REGION Network 64: **** 5.2 - Flow Equations **** Send Alarm If No Other Requests Is Active
   // Send Alarm If No Other Requests Is Active
   IF #SendAlarm[9] THEN
       #ReqSendToVDAlarm[9] := TRUE;   // SR flip-flop
   END_IF;
   IF #SendDoneVD THEN #ReqSendToVDAlarm[9] := FALSE; END_IF;
   IF #SendAlarm[9] THEN
       #_LDBCheckMZ8(I_DBNr := #C_AlarmDBMZ8, O_DBLength => #AlarmLength, O_DBNr => #AlarmPointer);   // "LDBCheck"
   END_IF;
   IF "TRUE" THEN
       #_LMDBToDBMZ8(I_CopyDB := #SendAlarm[9],   // "LMDBToDB"
                     I_SourceDB := #C_AlarmDBMZ8,
                     I_StartAddresSourceDB := 0,
                     I_DestDB := #C_AlarmCompareDBMZ8,
                     I_StartAddressDestDB := 0,
                     I_LenghtBytes := #AlarmLength);
   END_IF;
END_REGION

REGION Network 65: **** 5.2 - Flow Equations **** Filter
   // Filter
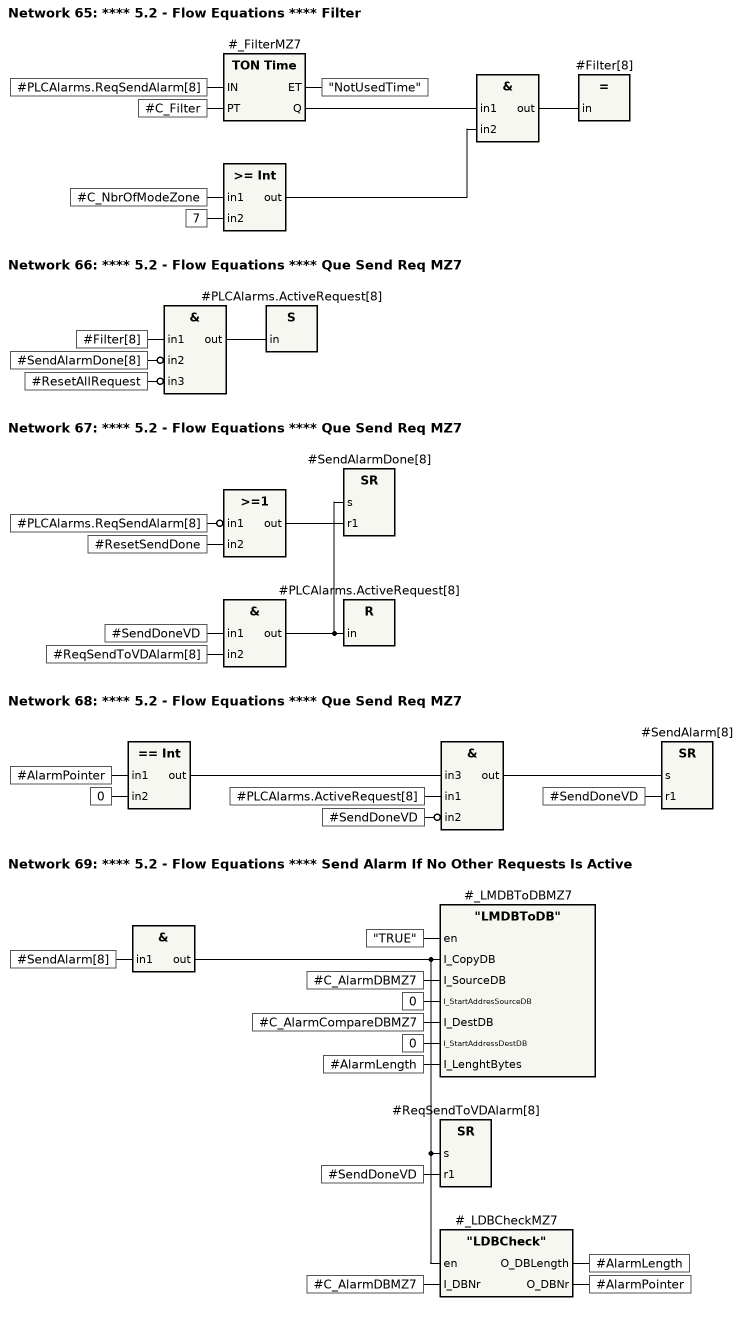
   #_FilterMZ7(IN := #PLCAlarms.ReqSendAlarm[8], PT := #C_Filter, ET => "NotUsedTime");   // TON
   #Filter[8] := #_FilterMZ7.Q AND (#C_NbrOfModeZone >= 7);
END_REGION

REGION Network 66: **** 5.2 - Flow Equations **** Que Send Req MZ7
   // Que Send Req
   IF #Filter[8] AND NOT #SendAlarmDone[8] AND NOT #ResetAllRequest THEN
       #PLCAlarms.ActiveRequest[8] := TRUE;
   END_IF;
END_REGION

REGION Network 67: **** 5.2 - Flow Equations **** Que Send Req MZ7
   // Que Send Req
   #_w1 := #SendDoneVD AND #ReqSendToVDAlarm[8];
   IF #_w1 THEN
       #SendAlarmDone[8] := TRUE;   // SR flip-flop
   END_IF;
   IF NOT #PLCAlarms.ReqSendAlarm[8] OR #ResetSendDone THEN #SendAlarmDone[8] := FALSE; END_IF;
   IF #_w1 THEN #PLCAlarms.ActiveRequest[8] := FALSE; END_IF;
END_REGION

REGION Network 68: **** 5.2 - Flow Equations **** Que Send Req MZ7
   // Que Send Req
   IF (#AlarmPointer = 0) AND #PLCAlarms.ActiveRequest[8] AND NOT #SendDoneVD THEN
       #SendAlarm[8] := TRUE;   // SR flip-flop
   END_IF;
   IF #SendDoneVD THEN #SendAlarm[8] := FALSE; END_IF;
END_REGION

REGION Network 69: **** 5.2 - Flow Equations **** Send Alarm If No Other Requests Is Active
   // Send Alarm If No Other Requests Is Active
   IF #SendAlarm[8] THEN
       #ReqSendToVDAlarm[8] := TRUE;   // SR flip-flop
   END_IF;
   IF #SendDoneVD THEN #ReqSendToVDAlarm[8] := FALSE; END_IF;
   IF #SendAlarm[8] THEN
       #_LDBCheckMZ7(I_DBNr := #C_AlarmDBMZ7, O_DBLength => #AlarmLength, O_DBNr => #AlarmPointer);   // "LDBCheck"
   END_IF;
   IF "TRUE" THEN
       #_LMDBToDBMZ7(I_CopyDB := #SendAlarm[8],   // "LMDBToDB"
                     I_SourceDB := #C_AlarmDBMZ7,
                     I_StartAddresSourceDB := 0,
                     I_DestDB := #C_AlarmCompareDBMZ7,
                     I_StartAddressDestDB := 0,
                     I_LenghtBytes := #AlarmLength);
   END_IF;
END_REGION

REGION Network 70: **** 5.2 - Flow Equations **** Filter
   // Filter
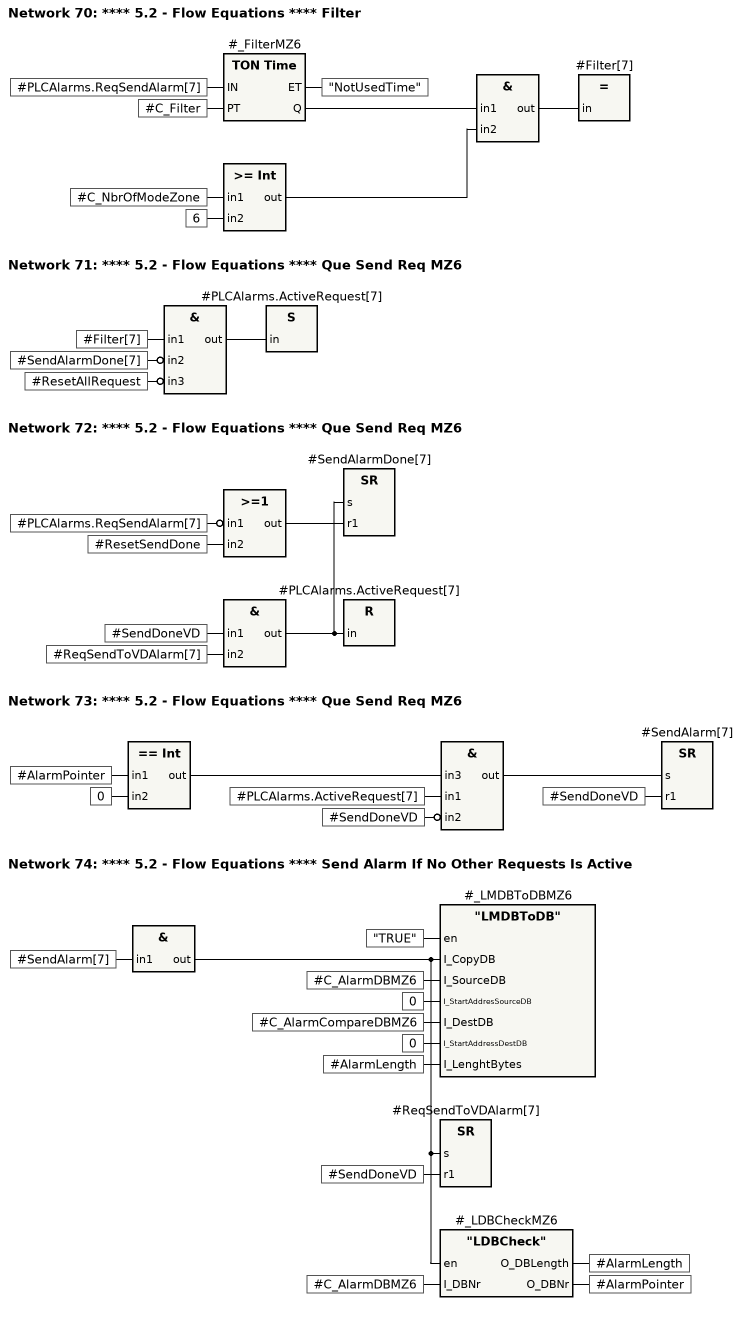
   #_FilterMZ6(IN := #PLCAlarms.ReqSendAlarm[7], PT := #C_Filter, ET => "NotUsedTime");   // TON
   #Filter[7] := #_FilterMZ6.Q AND (#C_NbrOfModeZone >= 6);
END_REGION

REGION Network 71: **** 5.2 - Flow Equations **** Que Send Req MZ6
   // Que Send Req
   IF #Filter[7] AND NOT #SendAlarmDone[7] AND NOT #ResetAllRequest THEN
       #PLCAlarms.ActiveRequest[7] := TRUE;
   END_IF;
END_REGION

REGION Network 72: **** 5.2 - Flow Equations **** Que Send Req MZ6
   // Que Send Req
   #_w1 := #SendDoneVD AND #ReqSendToVDAlarm[7];
   IF #_w1 THEN
       #SendAlarmDone[7] := TRUE;   // SR flip-flop
   END_IF;
   IF NOT #PLCAlarms.ReqSendAlarm[7] OR #ResetSendDone THEN #SendAlarmDone[7] := FALSE; END_IF;
   IF #_w1 THEN #PLCAlarms.ActiveRequest[7] := FALSE; END_IF;
END_REGION

REGION Network 73: **** 5.2 - Flow Equations **** Que Send Req MZ6
   // Que Send Req
   IF (#AlarmPointer = 0) AND #PLCAlarms.ActiveRequest[7] AND NOT #SendDoneVD THEN
       #SendAlarm[7] := TRUE;   // SR flip-flop
   END_IF;
   IF #SendDoneVD THEN #SendAlarm[7] := FALSE; END_IF;
END_REGION

REGION Network 74: **** 5.2 - Flow Equations **** Send Alarm If No Other Requests Is Active
   // Send Alarm If No Other Requests Is Active
   IF #SendAlarm[7] THEN
       #ReqSendToVDAlarm[7] := TRUE;   // SR flip-flop
   END_IF;
   IF #SendDoneVD THEN #ReqSendToVDAlarm[7] := FALSE; END_IF;
   IF #SendAlarm[7] THEN
       #_LDBCheckMZ6(I_DBNr := #C_AlarmDBMZ6, O_DBLength => #AlarmLength, O_DBNr => #AlarmPointer);   // "LDBCheck"
   END_IF;
   IF "TRUE" THEN
       #_LMDBToDBMZ6(I_CopyDB := #SendAlarm[7],   // "LMDBToDB"
                     I_SourceDB := #C_AlarmDBMZ6,
                     I_StartAddresSourceDB := 0,
                     I_DestDB := #C_AlarmCompareDBMZ6,
                     I_StartAddressDestDB := 0,
                     I_LenghtBytes := #AlarmLength);
   END_IF;
END_REGION

REGION Network 75: **** 5.2 - Flow Equations **** Filter
   // Filter
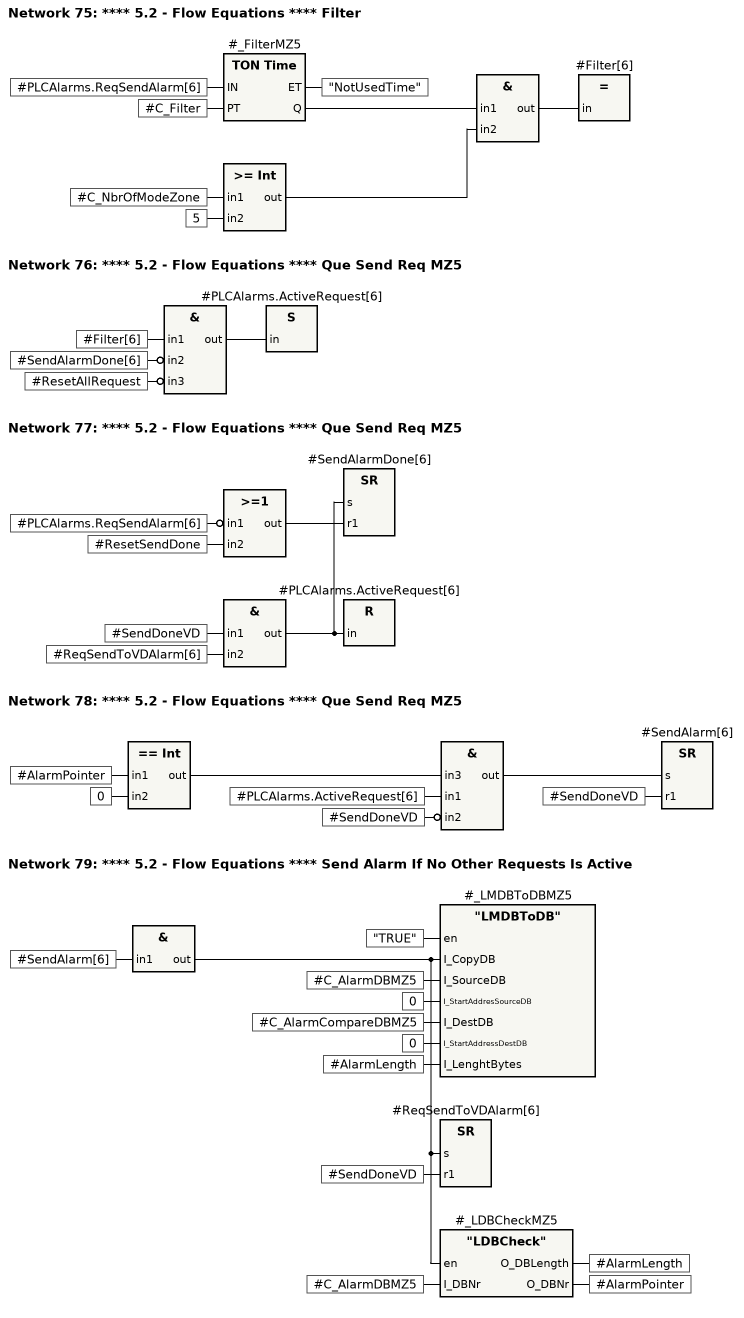
   #_FilterMZ5(IN := #PLCAlarms.ReqSendAlarm[6], PT := #C_Filter, ET => "NotUsedTime");   // TON
   #Filter[6] := #_FilterMZ5.Q AND (#C_NbrOfModeZone >= 5);
END_REGION

REGION Network 76: **** 5.2 - Flow Equations **** Que Send Req MZ5
   // Que Send Req
   IF #Filter[6] AND NOT #SendAlarmDone[6] AND NOT #ResetAllRequest THEN
       #PLCAlarms.ActiveRequest[6] := TRUE;
   END_IF;
END_REGION

REGION Network 77: **** 5.2 - Flow Equations **** Que Send Req MZ5
   // Que Send Req
   #_w1 := #SendDoneVD AND #ReqSendToVDAlarm[6];
   IF #_w1 THEN
       #SendAlarmDone[6] := TRUE;   // SR flip-flop
   END_IF;
   IF NOT #PLCAlarms.ReqSendAlarm[6] OR #ResetSendDone THEN #SendAlarmDone[6] := FALSE; END_IF;
   IF #_w1 THEN #PLCAlarms.ActiveRequest[6] := FALSE; END_IF;
END_REGION

REGION Network 78: **** 5.2 - Flow Equations **** Que Send Req MZ5
   // Que Send Req
   IF (#AlarmPointer = 0) AND #PLCAlarms.ActiveRequest[6] AND NOT #SendDoneVD THEN
       #SendAlarm[6] := TRUE;   // SR flip-flop
   END_IF;
   IF #SendDoneVD THEN #SendAlarm[6] := FALSE; END_IF;
END_REGION

REGION Network 79: **** 5.2 - Flow Equations **** Send Alarm If No Other Requests Is Active
   // Send Alarm If No Other Requests Is Active
   IF #SendAlarm[6] THEN
       #ReqSendToVDAlarm[6] := TRUE;   // SR flip-flop
   END_IF;
   IF #SendDoneVD THEN #ReqSendToVDAlarm[6] := FALSE; END_IF;
   IF #SendAlarm[6] THEN
       #_LDBCheckMZ5(I_DBNr := #C_AlarmDBMZ5, O_DBLength => #AlarmLength, O_DBNr => #AlarmPointer);   // "LDBCheck"
   END_IF;
   IF "TRUE" THEN
       #_LMDBToDBMZ5(I_CopyDB := #SendAlarm[6],   // "LMDBToDB"
                     I_SourceDB := #C_AlarmDBMZ5,
                     I_StartAddresSourceDB := 0,
                     I_DestDB := #C_AlarmCompareDBMZ5,
                     I_StartAddressDestDB := 0,
                     I_LenghtBytes := #AlarmLength);
   END_IF;
END_REGION

REGION Network 80: **** 5.2 - Flow Equations **** Filter
   // Filter
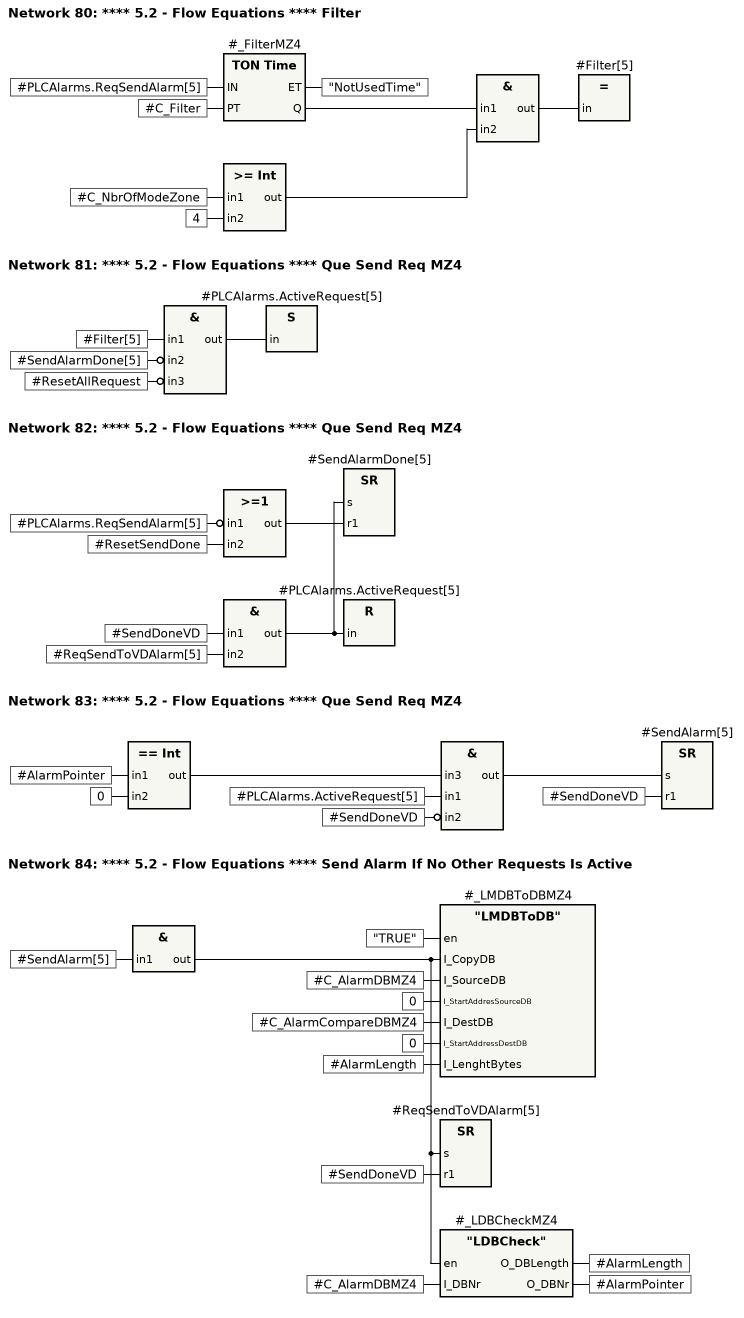
   #_FilterMZ4(IN := #PLCAlarms.ReqSendAlarm[5], PT := #C_Filter, ET => "NotUsedTime");   // TON
   #Filter[5] := #_FilterMZ4.Q AND (#C_NbrOfModeZone >= 4);
END_REGION

REGION Network 81: **** 5.2 - Flow Equations **** Que Send Req MZ4
   // Que Send Req
   IF #Filter[5] AND NOT #SendAlarmDone[5] AND NOT #ResetAllRequest THEN
       #PLCAlarms.ActiveRequest[5] := TRUE;
   END_IF;
END_REGION

REGION Network 82: **** 5.2 - Flow Equations **** Que Send Req MZ4
   // Que Send Req
   #_w1 := #SendDoneVD AND #ReqSendToVDAlarm[5];
   IF #_w1 THEN
       #SendAlarmDone[5] := TRUE;   // SR flip-flop
   END_IF;
   IF NOT #PLCAlarms.ReqSendAlarm[5] OR #ResetSendDone THEN #SendAlarmDone[5] := FALSE; END_IF;
   IF #_w1 THEN #PLCAlarms.ActiveRequest[5] := FALSE; END_IF;
END_REGION

REGION Network 83: **** 5.2 - Flow Equations **** Que Send Req MZ4
   // Que Send Req
   IF (#AlarmPointer = 0) AND #PLCAlarms.ActiveRequest[5] AND NOT #SendDoneVD THEN
       #SendAlarm[5] := TRUE;   // SR flip-flop
   END_IF;
   IF #SendDoneVD THEN #SendAlarm[5] := FALSE; END_IF;
END_REGION

REGION Network 84: **** 5.2 - Flow Equations **** Send Alarm If No Other Requests Is Active
   // Send Alarm If No Other Requests Is Active
   IF #SendAlarm[5] THEN
       #ReqSendToVDAlarm[5] := TRUE;   // SR flip-flop
   END_IF;
   IF #SendDoneVD THEN #ReqSendToVDAlarm[5] := FALSE; END_IF;
   IF #SendAlarm[5] THEN
       #_LDBCheckMZ4(I_DBNr := #C_AlarmDBMZ4, O_DBLength => #AlarmLength, O_DBNr => #AlarmPointer);   // "LDBCheck"
   END_IF;
   IF "TRUE" THEN
       #_LMDBToDBMZ4(I_CopyDB := #SendAlarm[5],   // "LMDBToDB"
                     I_SourceDB := #C_AlarmDBMZ4,
                     I_StartAddresSourceDB := 0,
                     I_DestDB := #C_AlarmCompareDBMZ4,
                     I_StartAddressDestDB := 0,
                     I_LenghtBytes := #AlarmLength);
   END_IF;
END_REGION

REGION Network 85: **** 5.2 - Flow Equations **** Filter
   // Filter
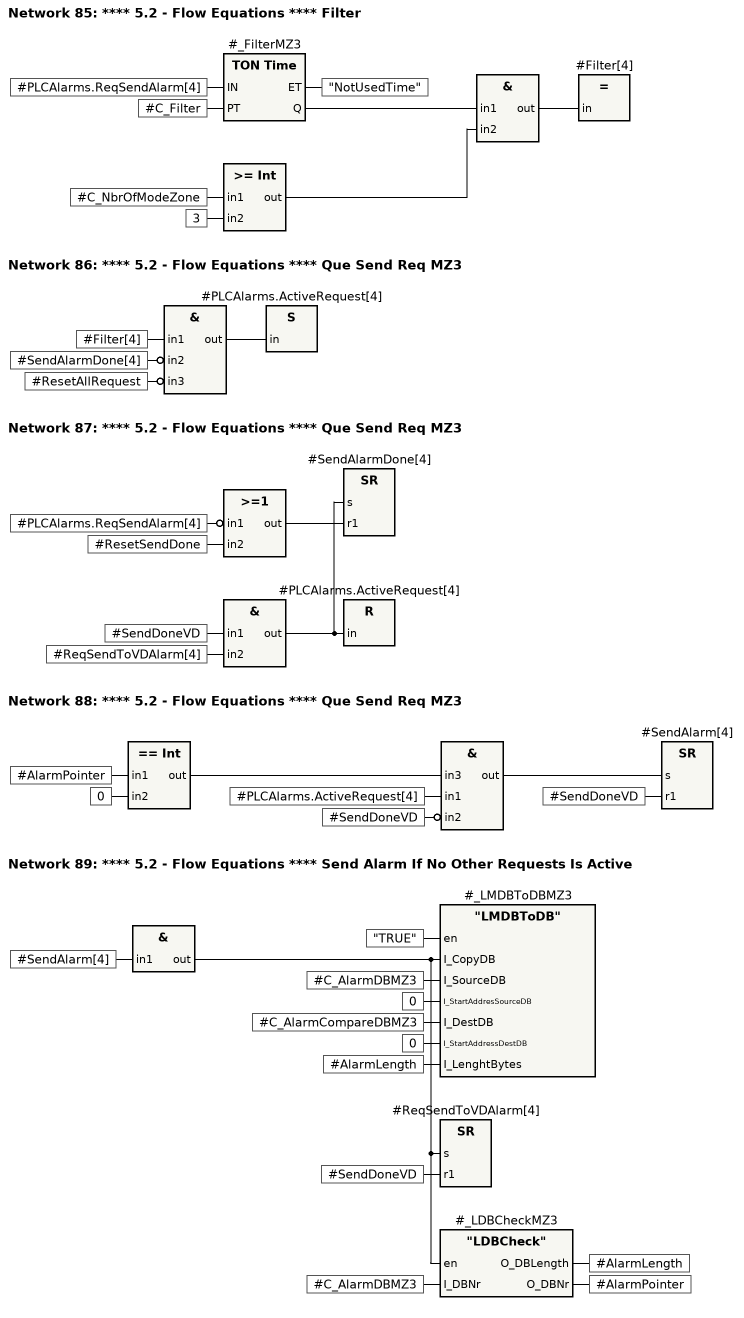
   #_FilterMZ3(IN := #PLCAlarms.ReqSendAlarm[4], PT := #C_Filter, ET => "NotUsedTime");   // TON
   #Filter[4] := #_FilterMZ3.Q AND (#C_NbrOfModeZone >= 3);
END_REGION

REGION Network 86: **** 5.2 - Flow Equations **** Que Send Req MZ3
   // Que Send Req
   IF #Filter[4] AND NOT #SendAlarmDone[4] AND NOT #ResetAllRequest THEN
       #PLCAlarms.ActiveRequest[4] := TRUE;
   END_IF;
END_REGION

REGION Network 87: **** 5.2 - Flow Equations **** Que Send Req MZ3
   // Que Send Req
   #_w1 := #SendDoneVD AND #ReqSendToVDAlarm[4];
   IF #_w1 THEN
       #SendAlarmDone[4] := TRUE;   // SR flip-flop
   END_IF;
   IF NOT #PLCAlarms.ReqSendAlarm[4] OR #ResetSendDone THEN #SendAlarmDone[4] := FALSE; END_IF;
   IF #_w1 THEN #PLCAlarms.ActiveRequest[4] := FALSE; END_IF;
END_REGION

REGION Network 88: **** 5.2 - Flow Equations **** Que Send Req MZ3
   // Que Send Req
   IF (#AlarmPointer = 0) AND #PLCAlarms.ActiveRequest[4] AND NOT #SendDoneVD THEN
       #SendAlarm[4] := TRUE;   // SR flip-flop
   END_IF;
   IF #SendDoneVD THEN #SendAlarm[4] := FALSE; END_IF;
END_REGION

REGION Network 89: **** 5.2 - Flow Equations **** Send Alarm If No Other Requests Is Active
   // Send Alarm If No Other Requests Is Active
   IF #SendAlarm[4] THEN
       #ReqSendToVDAlarm[4] := TRUE;   // SR flip-flop
   END_IF;
   IF #SendDoneVD THEN #ReqSendToVDAlarm[4] := FALSE; END_IF;
   IF #SendAlarm[4] THEN
       #_LDBCheckMZ3(I_DBNr := #C_AlarmDBMZ3, O_DBLength => #AlarmLength, O_DBNr => #AlarmPointer);   // "LDBCheck"
   END_IF;
   IF "TRUE" THEN
       #_LMDBToDBMZ3(I_CopyDB := #SendAlarm[4],   // "LMDBToDB"
                     I_SourceDB := #C_AlarmDBMZ3,
                     I_StartAddresSourceDB := 0,
                     I_DestDB := #C_AlarmCompareDBMZ3,
                     I_StartAddressDestDB := 0,
                     I_LenghtBytes := #AlarmLength);
   END_IF;
END_REGION

REGION Network 90: **** 5.2 - Flow Equations **** Filter
   // Filter
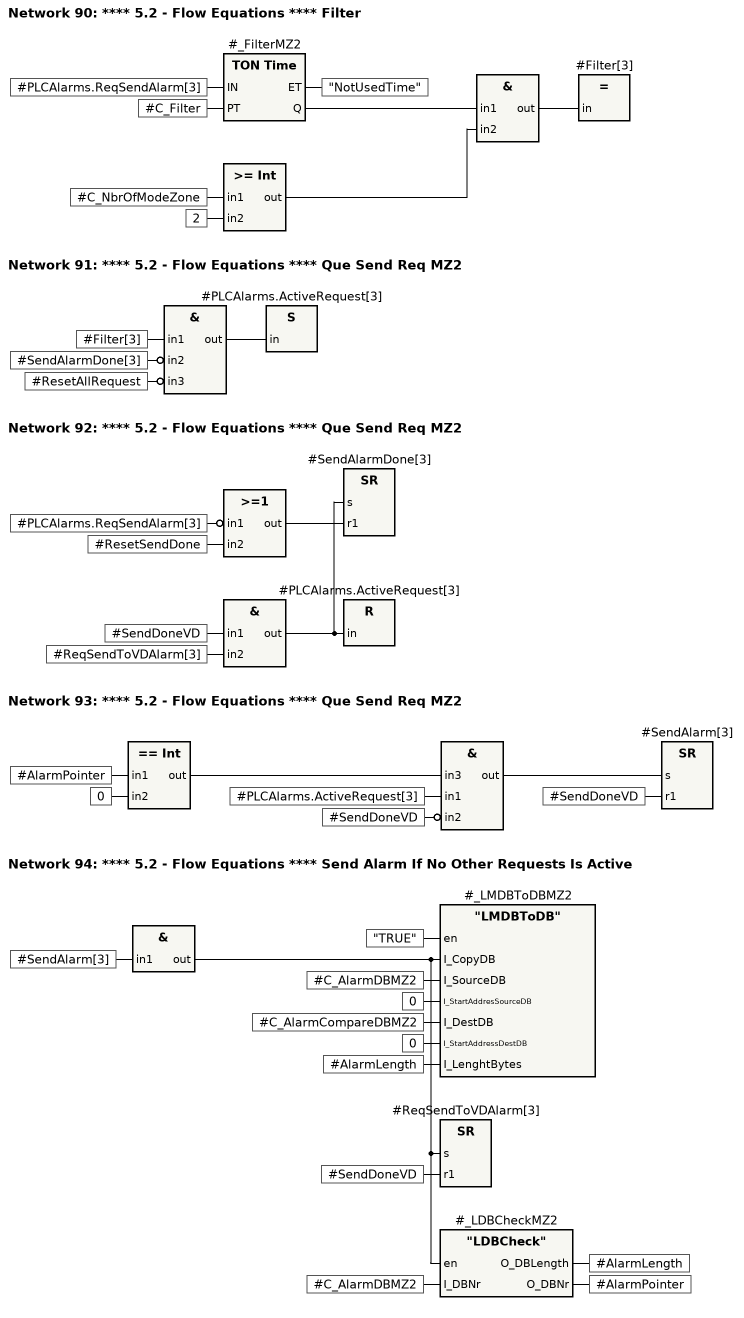
   #_FilterMZ2(IN := #PLCAlarms.ReqSendAlarm[3], PT := #C_Filter, ET => "NotUsedTime");   // TON
   #Filter[3] := #_FilterMZ2.Q AND (#C_NbrOfModeZone >= 2);
END_REGION

REGION Network 91: **** 5.2 - Flow Equations **** Que Send Req MZ2
   // Que Send Req
   IF #Filter[3] AND NOT #SendAlarmDone[3] AND NOT #ResetAllRequest THEN
       #PLCAlarms.ActiveRequest[3] := TRUE;
   END_IF;
END_REGION

REGION Network 92: **** 5.2 - Flow Equations **** Que Send Req MZ2
   // Que Send Req
   #_w1 := #SendDoneVD AND #ReqSendToVDAlarm[3];
   IF #_w1 THEN
       #SendAlarmDone[3] := TRUE;   // SR flip-flop
   END_IF;
   IF NOT #PLCAlarms.ReqSendAlarm[3] OR #ResetSendDone THEN #SendAlarmDone[3] := FALSE; END_IF;
   IF #_w1 THEN #PLCAlarms.ActiveRequest[3] := FALSE; END_IF;
END_REGION

REGION Network 93: **** 5.2 - Flow Equations **** Que Send Req MZ2
   // Que Send Req
   IF (#AlarmPointer = 0) AND #PLCAlarms.ActiveRequest[3] AND NOT #SendDoneVD THEN
       #SendAlarm[3] := TRUE;   // SR flip-flop
   END_IF;
   IF #SendDoneVD THEN #SendAlarm[3] := FALSE; END_IF;
END_REGION

REGION Network 94: **** 5.2 - Flow Equations **** Send Alarm If No Other Requests Is Active
   // Send Alarm If No Other Requests Is Active
   IF #SendAlarm[3] THEN
       #ReqSendToVDAlarm[3] := TRUE;   // SR flip-flop
   END_IF;
   IF #SendDoneVD THEN #ReqSendToVDAlarm[3] := FALSE; END_IF;
   IF #SendAlarm[3] THEN
       #_LDBCheckMZ2(I_DBNr := #C_AlarmDBMZ2, O_DBLength => #AlarmLength, O_DBNr => #AlarmPointer);   // "LDBCheck"
   END_IF;
   IF "TRUE" THEN
       #_LMDBToDBMZ2(I_CopyDB := #SendAlarm[3],   // "LMDBToDB"
                     I_SourceDB := #C_AlarmDBMZ2,
                     I_StartAddresSourceDB := 0,
                     I_DestDB := #C_AlarmCompareDBMZ2,
                     I_StartAddressDestDB := 0,
                     I_LenghtBytes := #AlarmLength);
   END_IF;
END_REGION

REGION Network 95: **** 5.2 - Flow Equations **** Filter
   // Filter
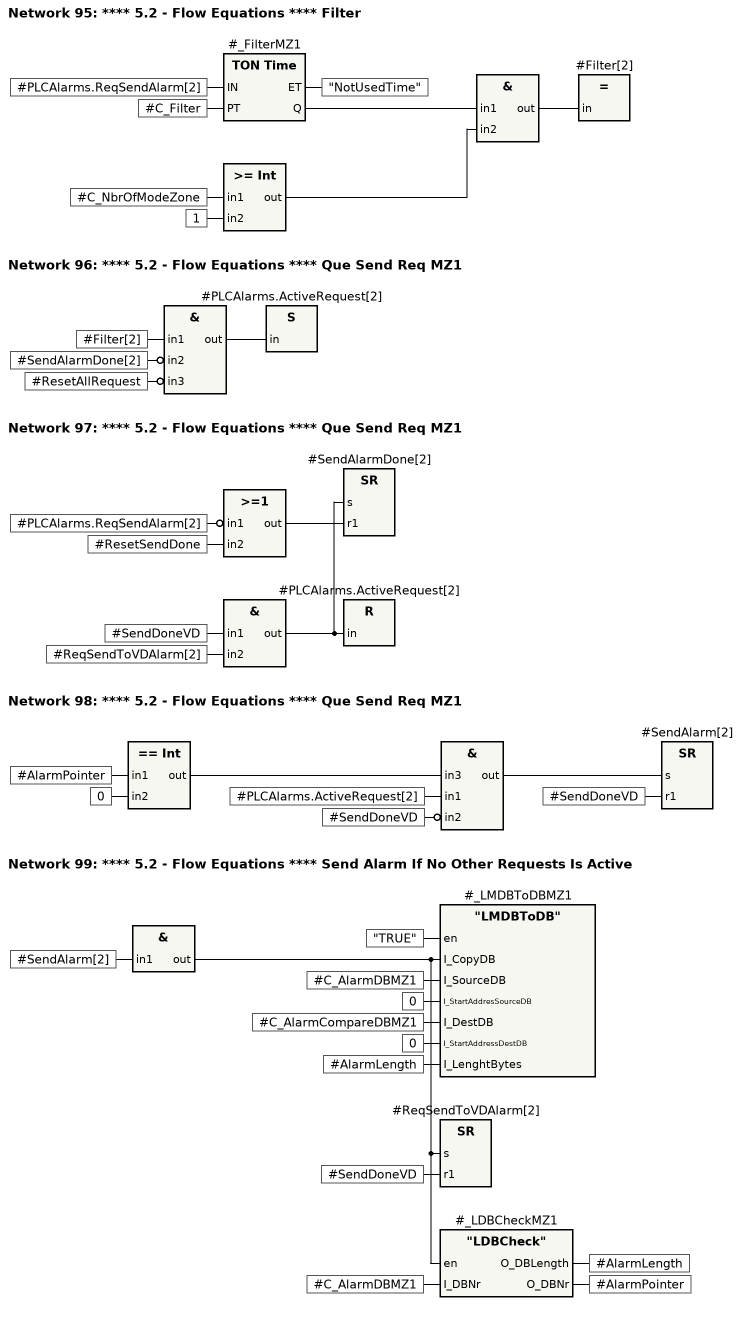
   #_FilterMZ1(IN := #PLCAlarms.ReqSendAlarm[2], PT := #C_Filter, ET => "NotUsedTime");   // TON
   #Filter[2] := #_FilterMZ1.Q AND (#C_NbrOfModeZone >= 1);
END_REGION

REGION Network 96: **** 5.2 - Flow Equations **** Que Send Req MZ1
   // Que Send Req
   IF #Filter[2] AND NOT #SendAlarmDone[2] AND NOT #ResetAllRequest THEN
       #PLCAlarms.ActiveRequest[2] := TRUE;
   END_IF;
END_REGION

REGION Network 97: **** 5.2 - Flow Equations **** Que Send Req MZ1
   // Que Send Req
   #_w1 := #SendDoneVD AND #ReqSendToVDAlarm[2];
   IF #_w1 THEN
       #SendAlarmDone[2] := TRUE;   // SR flip-flop
   END_IF;
   IF NOT #PLCAlarms.ReqSendAlarm[2] OR #ResetSendDone THEN #SendAlarmDone[2] := FALSE; END_IF;
   IF #_w1 THEN #PLCAlarms.ActiveRequest[2] := FALSE; END_IF;
END_REGION

REGION Network 98: **** 5.2 - Flow Equations **** Que Send Req MZ1
   // Que Send Req
   IF (#AlarmPointer = 0) AND #PLCAlarms.ActiveRequest[2] AND NOT #SendDoneVD THEN
       #SendAlarm[2] := TRUE;   // SR flip-flop
   END_IF;
   IF #SendDoneVD THEN #SendAlarm[2] := FALSE; END_IF;
END_REGION

REGION Network 99: **** 5.2 - Flow Equations **** Send Alarm If No Other Requests Is Active
   // Send Alarm If No Other Requests Is Active
   IF #SendAlarm[2] THEN
       #ReqSendToVDAlarm[2] := TRUE;   // SR flip-flop
   END_IF;
   IF #SendDoneVD THEN #ReqSendToVDAlarm[2] := FALSE; END_IF;
   IF #SendAlarm[2] THEN
       #_LDBCheckMZ1(I_DBNr := #C_AlarmDBMZ1, O_DBLength => #AlarmLength, O_DBNr => #AlarmPointer);   // "LDBCheck"
   END_IF;
   IF "TRUE" THEN
       #_LMDBToDBMZ1(I_CopyDB := #SendAlarm[2],   // "LMDBToDB"
                     I_SourceDB := #C_AlarmDBMZ1,
                     I_StartAddresSourceDB := 0,
                     I_DestDB := #C_AlarmCompareDBMZ1,
                     I_StartAddressDestDB := 0,
                     I_LenghtBytes := #AlarmLength);
   END_IF;
END_REGION

REGION Network 100: **** 5.2 - Flow Equations **** Filter
   // Filter
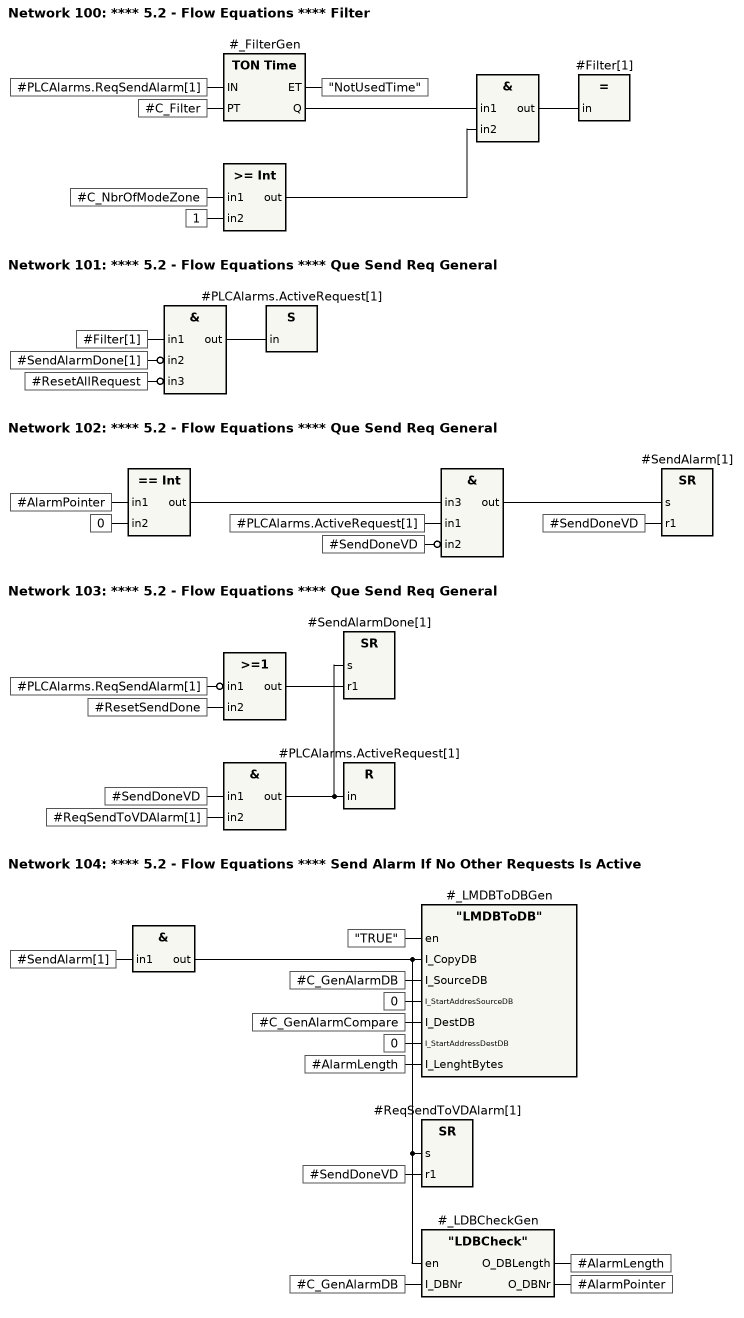
   #_FilterGen(IN := #PLCAlarms.ReqSendAlarm[1], PT := #C_Filter, ET => "NotUsedTime");   // TON
   #Filter[1] := #_FilterGen.Q AND (#C_NbrOfModeZone >= 1);
END_REGION

REGION Network 101: **** 5.2 - Flow Equations **** Que Send Req General
   // Que Send Req
   IF #Filter[1] AND NOT #SendAlarmDone[1] AND NOT #ResetAllRequest THEN
       #PLCAlarms.ActiveRequest[1] := TRUE;
   END_IF;
END_REGION

REGION Network 102: **** 5.2 - Flow Equations **** Que Send Req General
   // Que Send Req
   IF (#AlarmPointer = 0) AND #PLCAlarms.ActiveRequest[1] AND NOT #SendDoneVD THEN
       #SendAlarm[1] := TRUE;   // SR flip-flop
   END_IF;
   IF #SendDoneVD THEN #SendAlarm[1] := FALSE; END_IF;
END_REGION

REGION Network 103: **** 5.2 - Flow Equations **** Que Send Req General
   // Que Send Req
   #_w1 := #SendDoneVD AND #ReqSendToVDAlarm[1];
   IF #_w1 THEN
       #SendAlarmDone[1] := TRUE;   // SR flip-flop
   END_IF;
   IF NOT #PLCAlarms.ReqSendAlarm[1] OR #ResetSendDone THEN #SendAlarmDone[1] := FALSE; END_IF;
   IF #_w1 THEN #PLCAlarms.ActiveRequest[1] := FALSE; END_IF;
END_REGION

REGION Network 104: **** 5.2 - Flow Equations **** Send Alarm If No Other Requests Is Active
   // Send Alarm If No Other Requests Is Active
   IF #SendAlarm[1] THEN
       #ReqSendToVDAlarm[1] := TRUE;   // SR flip-flop
   END_IF;
   IF #SendDoneVD THEN #ReqSendToVDAlarm[1] := FALSE; END_IF;
   IF #SendAlarm[1] THEN
       #_LDBCheckGen(I_DBNr := #C_GenAlarmDB, O_DBLength => #AlarmLength, O_DBNr => #AlarmPointer);   // "LDBCheck"
   END_IF;
   IF "TRUE" THEN
       #_LMDBToDBGen(I_CopyDB := #SendAlarm[1],   // "LMDBToDB"
                     I_SourceDB := #C_GenAlarmDB,
                     I_StartAddresSourceDB := 0,
                     I_DestDB := #C_GenAlarmCompare,
                     I_StartAddressDestDB := 0,
                     I_LenghtBytes := #AlarmLength);
   END_IF;
END_REGION
END_FUNCTION_BLOCK

FUNCTION_BLOCK "LDBCheck"   // FB2146, FBD
TITLE = LDBCheck
{ S7_Optimized_Access := 'FALSE' }
AUTHOR : VCC
FAMILY : DataHand
VERSION : 0.1
// =============================================================================
// This Module Checks DB Length & DB Number
// =============================================================================
// stored: AutoNumber false, IsIECCheckEnabled true, SetENOAutomatically False, UDAEnableTagReadback false
   VAR_INPUT
      I_DBNr { ExternalAccessible := 'False'; ExternalVisible := 'False'; ExternalWritable := 'False'} : DB_ANY;   // DB
   END_VAR
   VAR_OUTPUT
      O_DBLength { ExternalAccessible := 'False'; ExternalVisible := 'False'; ExternalWritable := 'False'} : Word;   // DB Length
      O_DBNr { ExternalAccessible := 'False'; ExternalVisible := 'False'; ExternalWritable := 'False'} : Word;   // DB Nr
   END_VAR
BEGIN

NETWORK
TITLE = **** 5.2 - Equations - Flow Equations **** Load DB Number & Number
// Load DB Length & Number
      OPN   #I_DBNr;
      L     DBLG;
      T     #O_DBLength;
      L     DBNO;
      T     #O_DBNr;
END_FUNCTION_BLOCK

FUNCTION_BLOCK "LMDBToDB"   // FB2145, FBD
TITLE = LMDBToDB
{ S7_Optimized_Access := 'FALSE' }
AUTHOR : VCC
FAMILY : DataHand
VERSION : 0.1
// =============================================================================
// This module Copies data from DB to DB
// =============================================================================
// stored: AutoNumber false, IsIECCheckEnabled true, SetENOAutomatically False, UDAEnableTagReadback false
   VAR_INPUT
      I_CopyDB { ExternalAccessible := 'False'; ExternalVisible := 'False'; ExternalWritable := 'False'} : Bool;   // Copy DB
      I_SourceDB { ExternalAccessible := 'False'; ExternalVisible := 'False'; ExternalWritable := 'False'} : DB_ANY;   // Source DB
      I_StartAddresSourceDB { ExternalAccessible := 'False'; ExternalVisible := 'False'; ExternalWritable := 'False'} : Int;   // Address
      I_DestDB { ExternalAccessible := 'False'; ExternalVisible := 'False'; ExternalWritable := 'False'} : DB_ANY;   // Dest DB
      I_StartAddressDestDB { ExternalAccessible := 'False'; ExternalVisible := 'False'; ExternalWritable := 'False'} : Int;   // Address
      I_LenghtBytes { ExternalAccessible := 'False'; ExternalVisible := 'False'; ExternalWritable := 'False'} : Word;   // Length
   END_VAR
   VAR_TEMP
      SourcePointer : Any;   // Temp
      DestPointer : Any;   // Temp
      SourceDB : Int;   // Temp
      DestDB : Int;   // Temp
   END_VAR
BEGIN

NETWORK
TITLE = **** 1 - Inputs **** DB Pointers
// DB Pointers
      OPN   #I_SourceDB;
      L     DBNO;
      T     #SourceDB;
      OPN   #I_DestDB;
      L     DBNO;
      T     #DestDB;

NETWORK
TITLE = **** 5.2 - Equations - Flow Equations **** Load Pointers
// Load Pointers
// APa Cleaning Warnings
      A     #I_CopyDB;
      JCN   ncAp;
      LAR1  P##SourcePointer;
      L     16#1002;
      T     LW [AR1, P#0.0];
      L     #I_LenghtBytes;
      T     LW [AR1, P#2.0];
      L     #SourceDB;
      T     LW [AR1, P#4.0];
      L     #I_StartAddresSourceDB;
      SLD   3;
      OD    16#8400_0000;
      T     LD [AR1, P#6.0];
      LAR1  P##DestPointer;
      L     16#1002;
      T     LW [AR1, P#0.0];
      L     #I_LenghtBytes;
      T     LW [AR1, P#2.0];
      L     #DestDB;
      T     LW [AR1, P#4.0];
      L     #I_StartAddressDestDB;
      SLD   3;
      OD    16#8400_0000;
      T     LD [AR1, P#6.0];
//      L     16#1002
//      T     %LW10
//      L     #I_LenghtBytes
//      T     %LW12
//      L     #DestDB
//      T     %LW14
//      L     #I_StartAddressDestDB
//      SLD   3
//      OD    16#8400_0000
//      T     %LD16
      CALL  BLKMOV
      ( SRCBLK  := #SourcePointer,
        RET_VAL := "NotUsedInt",
        DSTBLK  := #DestPointer
      );
ncAp: NOP   0;
END_FUNCTION_BLOCK

FUNCTION_BLOCK "LMovFnc2Pos2S"   // FB2162, FBD
TITLE = LMovFnc2Pos2S
{ S7_Optimized_Access := 'TRUE' }
AUTHOR : VCC
FAMILY : Tooling
VERSION : 0.1
// =============================================================================
// This module will be used for the steering of a two Position movement wit 2 speed
// It will get the commands from different Modes, evaluate the status of the 
// Interlock and give the command to the Actuator or direct to simple outputs.
// =============================================================================
// stored: AutoNumber false, IsIECCheckEnabled false, IsRetainMemResEnabled false, MemoryReserve 100, SetENOAutomatically False, UDAEnableTagReadback false
   VAR_INPUT
      I_PosSet { ExternalAccessible := 'False'; ExternalVisible := 'False'; ExternalWritable := 'False'} : Bool;   // Position Set detection or summary
      I_LowSpeedSetDet { ExternalAccessible := 'False'; ExternalVisible := 'False'; ExternalWritable := 'False'} : Bool;   // Slow Set detection or summary
      I_PosRes { ExternalAccessible := 'False'; ExternalVisible := 'False'; ExternalWritable := 'False'} : Bool;   // Position Reset detection or summary
      I_LowSpeedResDet { ExternalAccessible := 'False'; ExternalVisible := 'False'; ExternalWritable := 'False'} : Bool;   // Slow Reset detection or summary
      I_PBSet { ExternalAccessible := 'False'; ExternalVisible := 'False'; ExternalWritable := 'False'} : Bool;   // Push button for Set direction (used in manual with button OP panels )
      I_PBReset { ExternalAccessible := 'False'; ExternalVisible := 'False'; ExternalWritable := 'False'} : Bool;   // Push button for Reset direction (used in manual with Pushbutton OP panels)
      I_SetBegin { ExternalAccessible := 'False'; ExternalVisible := 'False'; ExternalWritable := 'False'} : Bool;   // Function Set begin selection
      I_ResBegin { ExternalAccessible := 'False'; ExternalVisible := 'False'; ExternalWritable := 'False'} : Bool;   // Function Reset begin selection
      I_SetIntlkOK { ExternalAccessible := 'False'; ExternalVisible := 'False'; ExternalWritable := 'False'} : Bool;   // Set Interlock
      I_ResIntlkOK { ExternalAccessible := 'False'; ExternalVisible := 'False'; ExternalWritable := 'False'} : Bool;   // Reset Interlock
      I_SafetyOk { ExternalAccessible := 'False'; ExternalVisible := 'False'; ExternalWritable := 'False'} : Bool;   // Safety Ok
      I_HardwareOk { ExternalAccessible := 'False'; ExternalVisible := 'False'; ExternalWritable := 'False'} : Bool;   // Safety Ok / Hardware Ok
   END_VAR
   VAR_OUTPUT
      O_CmdSetHighSpeed { ExternalAccessible := 'False'; ExternalVisible := 'False'; ExternalWritable := 'False'} : Bool;   // Command to Activate Set movement
      O_CmdResHighSpeed { ExternalAccessible := 'False'; ExternalVisible := 'False'; ExternalWritable := 'False'} : Bool;   // Command to Activate Reset movement
      O_CmdSetLowSpeed { ExternalAccessible := 'False'; ExternalVisible := 'False'; ExternalWritable := 'False'} : Bool;   // Command to Activate Slow Set movement
      O_CmdResLowSpeed { ExternalAccessible := 'False'; ExternalVisible := 'False'; ExternalWritable := 'False'} : Bool;   // Command to Activate Slow Reset movement
      O_CmdSet { ExternalAccessible := 'False'; ExternalVisible := 'False'; ExternalWritable := 'False'} : Bool;   // Command to activate Set movement / Command to Activate Set movement
      O_CmdRes { ExternalAccessible := 'False'; ExternalVisible := 'False'; ExternalWritable := 'False'} : Bool;   // Command to activate Reset movement / Command to Activate Reset movement
      O_FuncRunning { ExternalAccessible := 'False'; ExternalVisible := 'False'; ExternalWritable := 'False'} : Bool;   // Signal that the function is running
      O_FuncBusyTM { ExternalAccessible := 'False'; ExternalVisible := 'False'; ExternalWritable := 'False'} : Bool;   // Memory Signal that the function is busy
      O_SetFinished { ExternalAccessible := 'False'; ExternalVisible := 'False'; ExternalWritable := 'False'} : Bool;   // Function Set finished to Master Sequencing
      O_ResFinished { ExternalAccessible := 'False'; ExternalVisible := 'False'; ExternalWritable := 'False'} : Bool;   // Function Reset finished to Master Sequencing
      O_IntlkSetAlm { ExternalAccessible := 'False'; ExternalVisible := 'False'; ExternalWritable := 'False'} : Bool;   // Alarm Interlock Set
      O_IntlkResAlm { ExternalAccessible := 'False'; ExternalVisible := 'False'; ExternalWritable := 'False'} : Bool;   // Alarm Interlock Reset
      O_FuncIsSelInMan { ExternalAccessible := 'False'; ExternalVisible := 'False'; ExternalWritable := 'False'} : Bool;   // The function is Selected in manual Mode
      O_LED { ExternalAccessible := 'False'; ExternalVisible := 'False'; ExternalWritable := 'False'} : Bool;   // LED - Indication
      O_AlarmABCondition { ExternalAccessible := 'False'; ExternalVisible := 'False'; ExternalWritable := 'False'} : Bool;   // Alarms AB condition
   END_VAR
   VAR_IN_OUT
      IO_Modes : "Modes";   // Modes
      H_HMI : "H_HMI";   // Animation
      H_MovFnc2Pos2s : "H_MovFnc2Pos";   // Animation
      H_FncSelInHMI { ExternalAccessible := 'False'; ExternalVisible := 'False'; ExternalWritable := 'False'} : Bool;   // This function is Selected to run from HMI
      C_AlarmResetUsed { ExternalAccessible := 'False'; ExternalVisible := 'False'; ExternalWritable := 'False'} : Bool;   // If true, the alrms will be stored untill Reseted
      C_EnableMemBegin { ExternalAccessible := 'False'; ExternalVisible := 'False'; ExternalWritable := 'False'} : Bool;   // Enable memory Begin (Command request is memorised until pos reached)
      C_EnIntlkAlm { ExternalAccessible := 'False'; ExternalVisible := 'False'; ExternalWritable := 'False'} : Bool := TRUE;   // Enable Interlock Alarm
      C_ForceManual { ExternalAccessible := 'False'; ExternalVisible := 'False'; ExternalWritable := 'False'} : Bool := FALSE;   // Force Manual
   END_VAR
   VAR
      ResetAlarm { ExternalAccessible := 'False'; ExternalVisible := 'False'; ExternalWritable := 'False'} : Bool;   // Reset Alarm Memory
      CmdSetRequest { ExternalAccessible := 'False'; ExternalVisible := 'False'; ExternalWritable := 'False'} : Bool;   // Set Command request to Activate the Interlock
      CmdResRequest { ExternalAccessible := 'False'; ExternalVisible := 'False'; ExternalWritable := 'False'} : Bool;   // Reset Command request to Activate the Interlock
      EdgeStopDetSet { ExternalAccessible := 'False'; ExternalVisible := 'False'; ExternalWritable := 'False'} : Bool;   // Edge on stop detection to be abble to go over it in force manual
      EdgeStopDetRes { ExternalAccessible := 'False'; ExternalVisible := 'False'; ExternalWritable := 'False'} : Bool;   // Edge on stop detection to be abble to go over it in force manual
      IntlkSetAlm { ExternalAccessible := 'False'; ExternalVisible := 'False'; ExternalWritable := 'False'} : Bool;   // Alarm Interlock Set
      IntlkResAlm { ExternalAccessible := 'False'; ExternalVisible := 'False'; ExternalWritable := 'False'} : Bool;   // Alarm Interlock Reset
      CmdSet { ExternalAccessible := 'False'; ExternalVisible := 'False'; ExternalWritable := 'False'} : Bool;   // Command to Activate Set movement
      CmdSetSl { ExternalAccessible := 'False'; ExternalVisible := 'False'; ExternalWritable := 'False'} : Bool;   // Command to Activate Slow Set movement
      CmdRes { ExternalAccessible := 'False'; ExternalVisible := 'False'; ExternalWritable := 'False'} : Bool;   // Command to Activate Reset movement
      CmdResSl { ExternalAccessible := 'False'; ExternalVisible := 'False'; ExternalWritable := 'False'} : Bool;   // Command to Activate Slow Reset movement
      IntlkSetAlmCond { ExternalAccessible := 'False'; ExternalVisible := 'False'; ExternalWritable := 'False'} : Bool;   // Alarm Interlock Set condition
      IntlkResAlmCond { ExternalAccessible := 'False'; ExternalVisible := 'False'; ExternalWritable := 'False'} : Bool;   // Alarm Interlock Reset condition
      FuncRunning { ExternalAccessible := 'False'; ExternalVisible := 'False'; ExternalWritable := 'False'} : Bool;   // Function is running
      FuncBusyTM { ExternalAccessible := 'False'; ExternalVisible := 'False'; ExternalWritable := 'False'} : Bool;   // Memory Signal that the function is busy
      AlmFilterResult { ExternalAccessible := 'False'; ExternalVisible := 'False'; ExternalWritable := 'False'} : Bool;   // Alarm filter result
      _AlarmTimer { ExternalAccessible := 'False'; ExternalVisible := 'False'; ExternalWritable := 'False'} : "LTimer";
   END_VAR
   VAR_TEMP   // added for the SCL form of the ladder/FBD networks
      _w1 : Bool;
   END_VAR
BEGIN

REGION Network 1: **** 2.2 - Alarms - Alarm Generation **** Alarm Filter
   // Alarm Filter
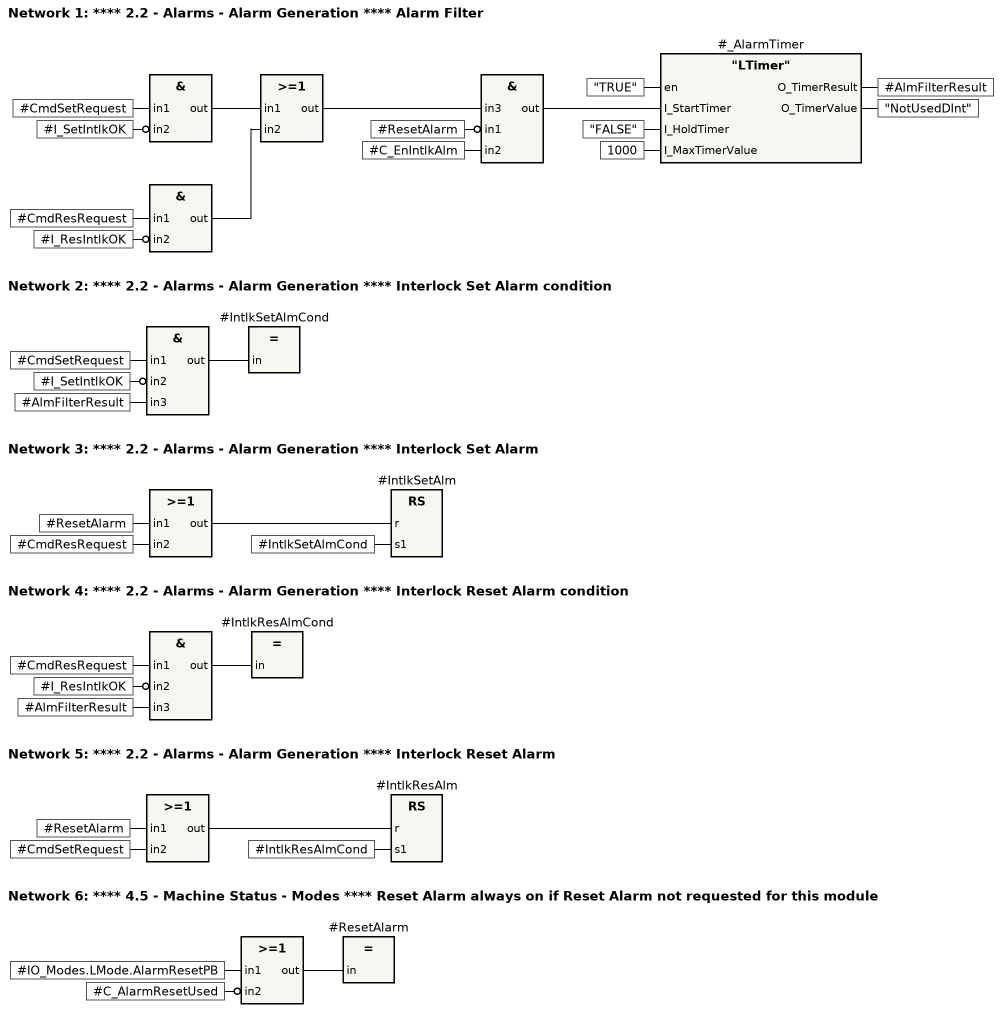
   IF "TRUE" THEN
       #_AlarmTimer(I_StartTimer := ((#CmdSetRequest AND NOT #I_SetIntlkOK) OR (#CmdResRequest AND NOT #I_ResIntlkOK)) AND NOT #ResetAlarm AND #C_EnIntlkAlm,   // "LTimer"
                    I_HoldTimer := "FALSE",
                    I_MaxTimerValue := 1000,
                    O_TimerResult => #AlmFilterResult,
                    O_TimerValue => "NotUsedDInt");
   END_IF;
END_REGION

REGION Network 2: **** 2.2 - Alarms - Alarm Generation **** Interlock Set Alarm condition
   // Interlock Set Alarm condition
   #IntlkSetAlmCond := #CmdSetRequest AND NOT #I_SetIntlkOK AND #AlmFilterResult;
END_REGION

REGION Network 3: **** 2.2 - Alarms - Alarm Generation **** Interlock Set Alarm
   // Interlock Set Alarm
   IF #ResetAlarm OR #CmdResRequest THEN
       #IntlkSetAlm := FALSE;   // RS flip-flop
   END_IF;
   IF #IntlkSetAlmCond THEN #IntlkSetAlm := TRUE; END_IF;
END_REGION

REGION Network 4: **** 2.2 - Alarms - Alarm Generation **** Interlock Reset Alarm condition
   // Interlock Reset Alarm condition
   #IntlkResAlmCond := #CmdResRequest AND NOT #I_ResIntlkOK AND #AlmFilterResult;
END_REGION

REGION Network 5: **** 2.2 - Alarms - Alarm Generation **** Interlock Reset Alarm
   // Interlock Reset Alarm
   IF #ResetAlarm OR #CmdSetRequest THEN
       #IntlkResAlm := FALSE;   // RS flip-flop
   END_IF;
   IF #IntlkResAlmCond THEN #IntlkResAlm := TRUE; END_IF;
END_REGION

REGION Network 6: **** 4.5 - Machine Status - Modes **** Reset Alarm always on if Reset Alarm not requested for this module
   // Reset Alarm always on if Reset Alarm not requested for this module
   #ResetAlarm := #IO_Modes.LMode.AlarmResetPB OR NOT #C_AlarmResetUsed;
END_REGION

REGION Network 7: **** 4.6 - Machine Status - Indication **** Icon Animation
   // Icon Animation
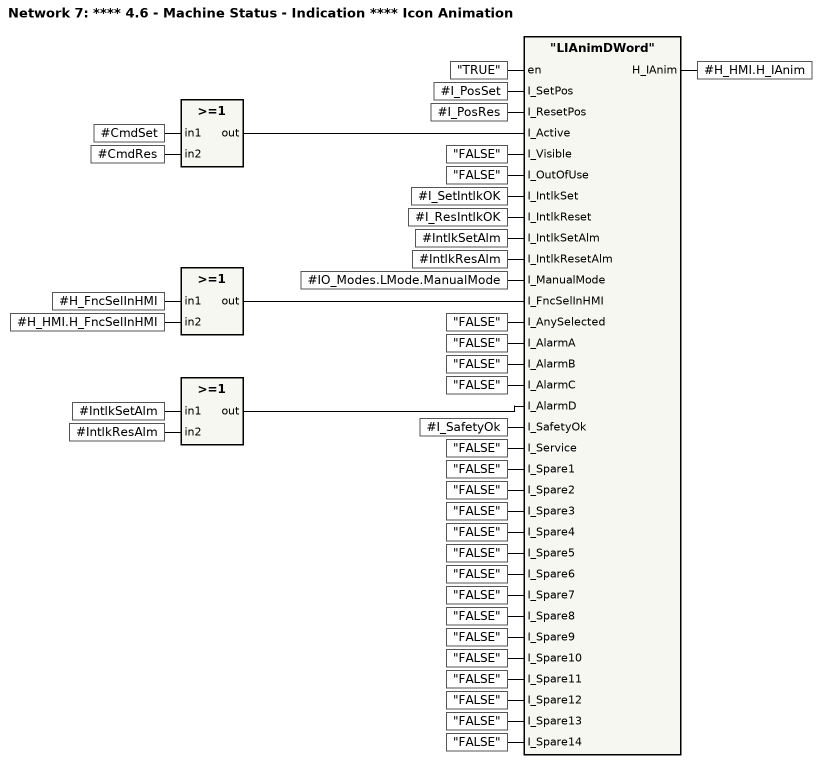
   IF "TRUE" THEN
       "LIAnimDWord"(I_SetPos := #I_PosSet,
                     I_ResetPos := #I_PosRes,
                     I_Active := #CmdSet OR #CmdRes,
                     I_Visible := "FALSE",
                     I_OutOfUse := "FALSE",
                     I_IntlkSet := #I_SetIntlkOK,
                     I_IntlkReset := #I_ResIntlkOK,
                     I_IntlkSetAlm := #IntlkSetAlm,
                     I_IntlkResetAlm := #IntlkResAlm,
                     I_ManualMode := #IO_Modes.LMode.ManualMode,
                     I_FncSelInHMI := #H_FncSelInHMI OR #H_HMI.H_FncSelInHMI,
                     I_AnySelected := "FALSE",
                     I_AlarmA := "FALSE",
                     I_AlarmB := "FALSE",
                     I_AlarmC := "FALSE",
                     I_AlarmD := #IntlkSetAlm OR #IntlkResAlm,
                     I_SafetyOk := #I_SafetyOk,
                     I_Service := "FALSE",
                     I_Spare1 := "FALSE",
                     I_Spare2 := "FALSE",
                     I_Spare3 := "FALSE",
                     I_Spare4 := "FALSE",
                     I_Spare5 := "FALSE",
                     I_Spare6 := "FALSE",
                     I_Spare7 := "FALSE",
                     I_Spare8 := "FALSE",
                     I_Spare9 := "FALSE",
                     I_Spare10 := "FALSE",
                     I_Spare11 := "FALSE",
                     I_Spare12 := "FALSE",
                     I_Spare13 := "FALSE",
                     I_Spare14 := "FALSE",
                     H_IAnim => #H_HMI.H_IAnim);
   END_IF;
END_REGION

REGION Network 8: **** 4.6 - Machine Status - Indication **** Animation
   // Animation
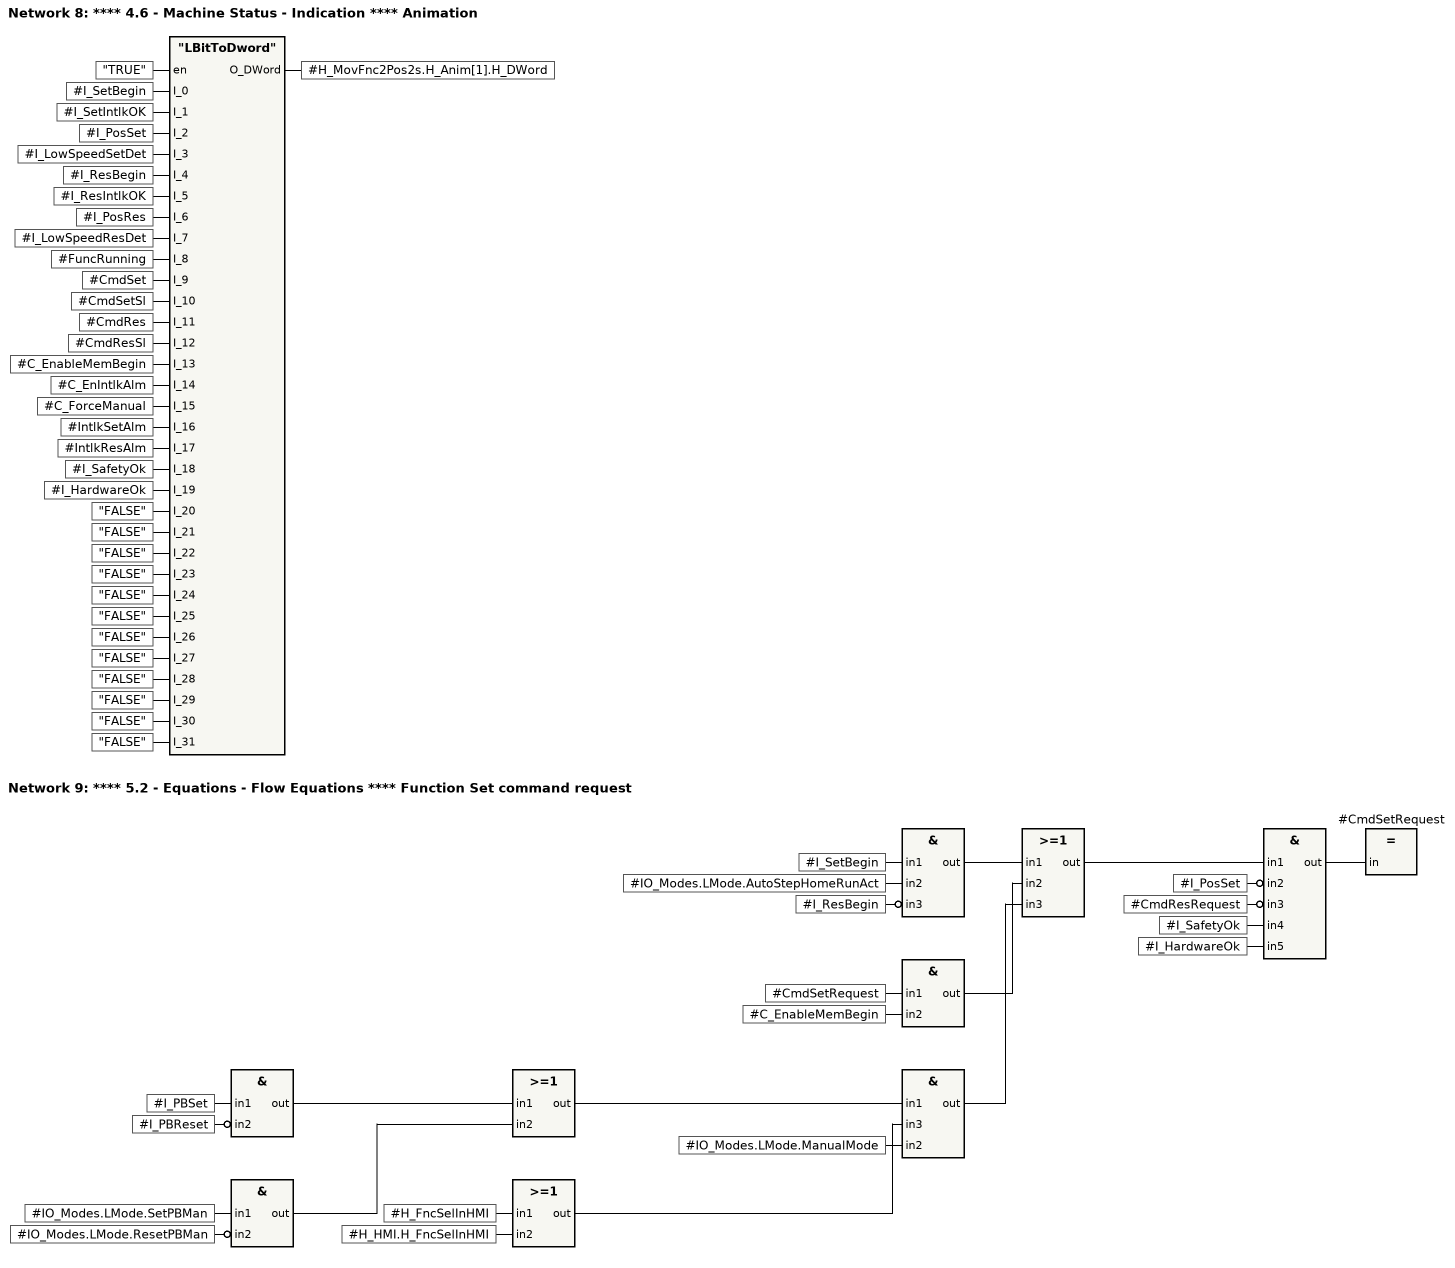
   IF "TRUE" THEN
       "LBitToDword"(I_0 := #I_SetBegin,
                     I_1 := #I_SetIntlkOK,
                     I_2 := #I_PosSet,
                     I_3 := #I_LowSpeedSetDet,
                     I_4 := #I_ResBegin,
                     I_5 := #I_ResIntlkOK,
                     I_6 := #I_PosRes,
                     I_7 := #I_LowSpeedResDet,
                     I_8 := #FuncRunning,
                     I_9 := #CmdSet,
                     I_10 := #CmdSetSl,
                     I_11 := #CmdRes,
                     I_12 := #CmdResSl,
                     I_13 := #C_EnableMemBegin,
                     I_14 := #C_EnIntlkAlm,
                     I_15 := #C_ForceManual,
                     I_16 := #IntlkSetAlm,
                     I_17 := #IntlkResAlm,
                     I_18 := #I_SafetyOk,
                     I_19 := #I_HardwareOk,
                     I_20 := "FALSE",
                     I_21 := "FALSE",
                     I_22 := "FALSE",
                     I_23 := "FALSE",
                     I_24 := "FALSE",
                     I_25 := "FALSE",
                     I_26 := "FALSE",
                     I_27 := "FALSE",
                     I_28 := "FALSE",
                     I_29 := "FALSE",
                     I_30 := "FALSE",
                     I_31 := "FALSE",
                     O_DWord => #H_MovFnc2Pos2s.H_Anim[1].H_DWord);
   END_IF;
END_REGION

REGION Network 9: **** 5.2 - Equations - Flow Equations **** Function Set command request
   // Function Set command request
   #CmdSetRequest := ((#I_SetBegin AND #IO_Modes.LMode.AutoStepHomeRunAct AND NOT #I_ResBegin) OR (#CmdSetRequest AND #C_EnableMemBegin) OR (((#I_PBSet AND NOT #I_PBReset) OR (#IO_Modes.LMode.SetPBMan AND NOT #IO_Modes.LMode.ResetPBMan)) AND (#H_FncSelInHMI OR #H_HMI.H_FncSelInHMI) AND #IO_Modes.LMode.ManualMode)) AND NOT #I_PosSet AND NOT #CmdResRequest AND #I_SafetyOk AND #I_HardwareOk;
END_REGION

REGION Network 10: **** 5.2 - Equations - Flow Equations **** Function Reset command request
   // Function Reset command request
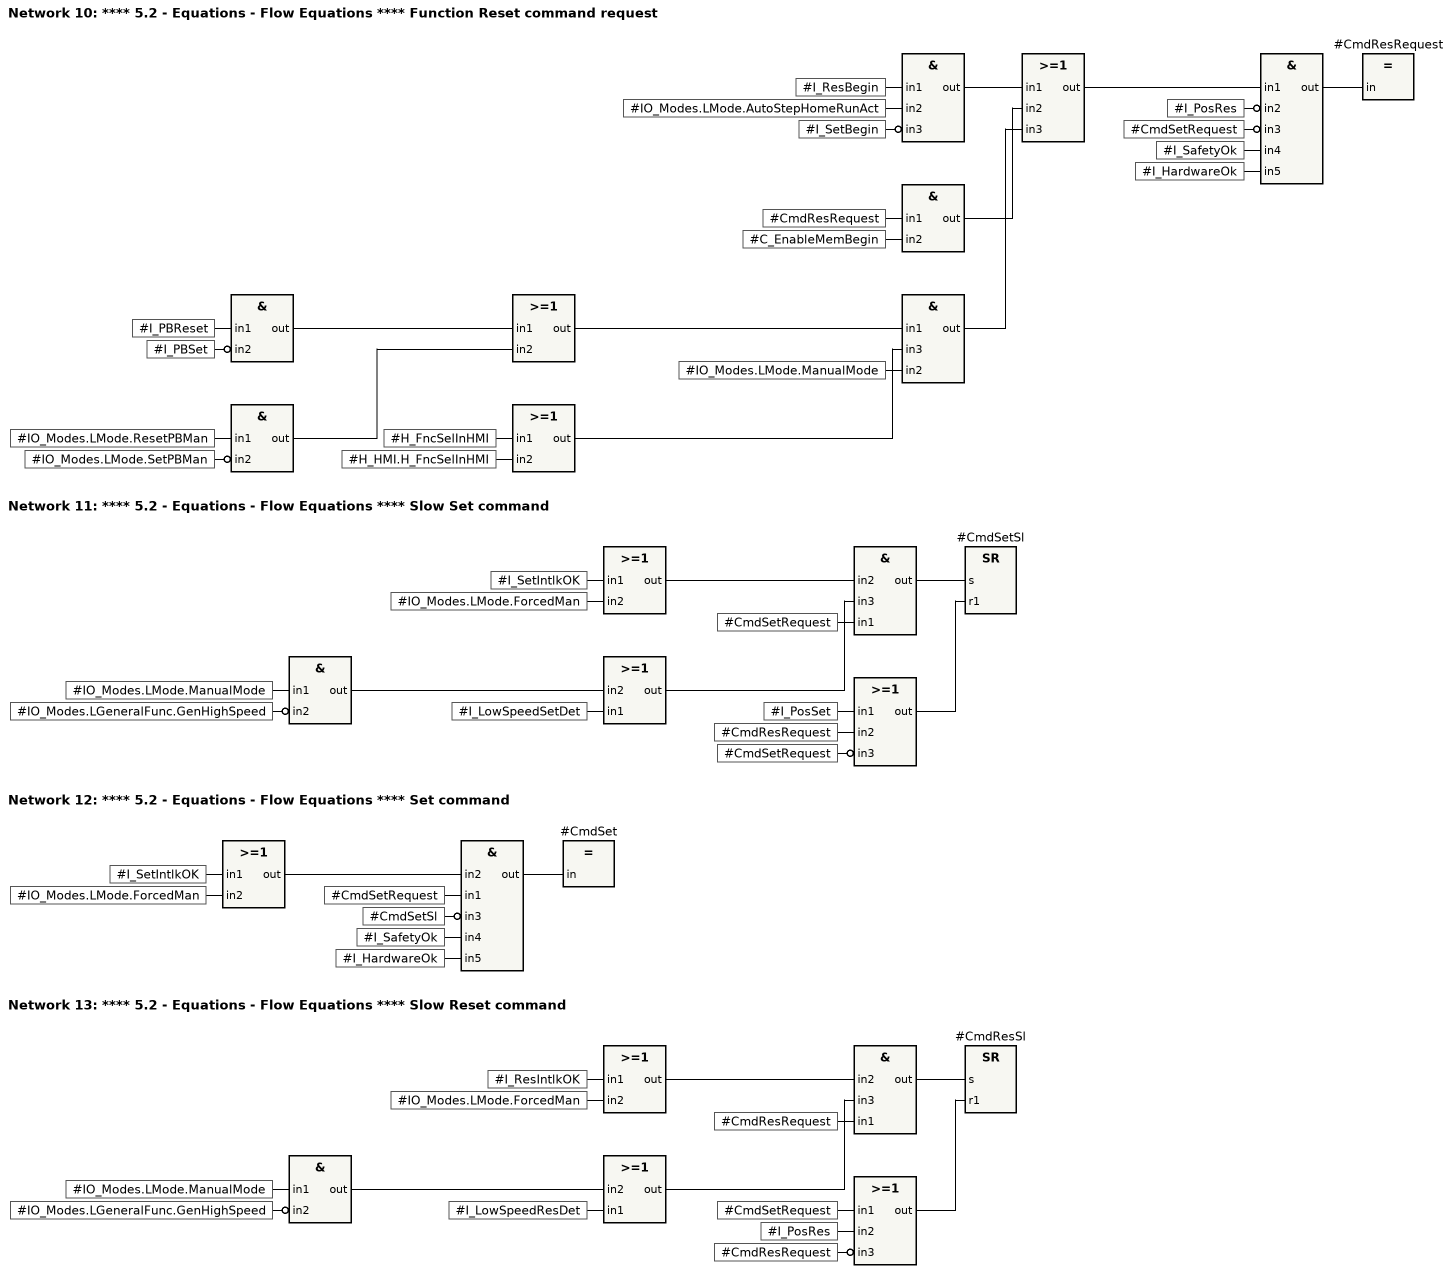
   #CmdResRequest := ((#I_ResBegin AND #IO_Modes.LMode.AutoStepHomeRunAct AND NOT #I_SetBegin) OR (#CmdResRequest AND #C_EnableMemBegin) OR (((#I_PBReset AND NOT #I_PBSet) OR (#IO_Modes.LMode.ResetPBMan AND NOT #IO_Modes.LMode.SetPBMan)) AND (#H_FncSelInHMI OR #H_HMI.H_FncSelInHMI) AND #IO_Modes.LMode.ManualMode)) AND NOT #I_PosRes AND NOT #CmdSetRequest AND #I_SafetyOk AND #I_HardwareOk;
END_REGION

REGION Network 11: **** 5.2 - Equations - Flow Equations **** Slow Set command
   // Slow Set command
   IF (#I_SetIntlkOK OR #IO_Modes.LMode.ForcedMan) AND ((#IO_Modes.LMode.ManualMode AND NOT #IO_Modes.LGeneralFunc.GenHighSpeed) OR #I_LowSpeedSetDet) AND #CmdSetRequest THEN
       #CmdSetSl := TRUE;   // SR flip-flop
   END_IF;
   IF #I_PosSet OR #CmdResRequest OR NOT #CmdSetRequest THEN #CmdSetSl := FALSE; END_IF;
END_REGION

REGION Network 12: **** 5.2 - Equations - Flow Equations **** Set command
   // Set command
   #CmdSet := (#I_SetIntlkOK OR #IO_Modes.LMode.ForcedMan) AND #CmdSetRequest AND NOT #CmdSetSl AND #I_SafetyOk AND #I_HardwareOk;
END_REGION

REGION Network 13: **** 5.2 - Equations - Flow Equations **** Slow Reset command
   // Slow Reset command
   IF (#I_ResIntlkOK OR #IO_Modes.LMode.ForcedMan) AND ((#IO_Modes.LMode.ManualMode AND NOT #IO_Modes.LGeneralFunc.GenHighSpeed) OR #I_LowSpeedResDet) AND #CmdResRequest THEN
       #CmdResSl := TRUE;   // SR flip-flop
   END_IF;
   IF #CmdSetRequest OR #I_PosRes OR NOT #CmdResRequest THEN #CmdResSl := FALSE; END_IF;
END_REGION

REGION Network 14: **** 5.2 - Equations - Flow Equations **** Reset command
   // Reset command
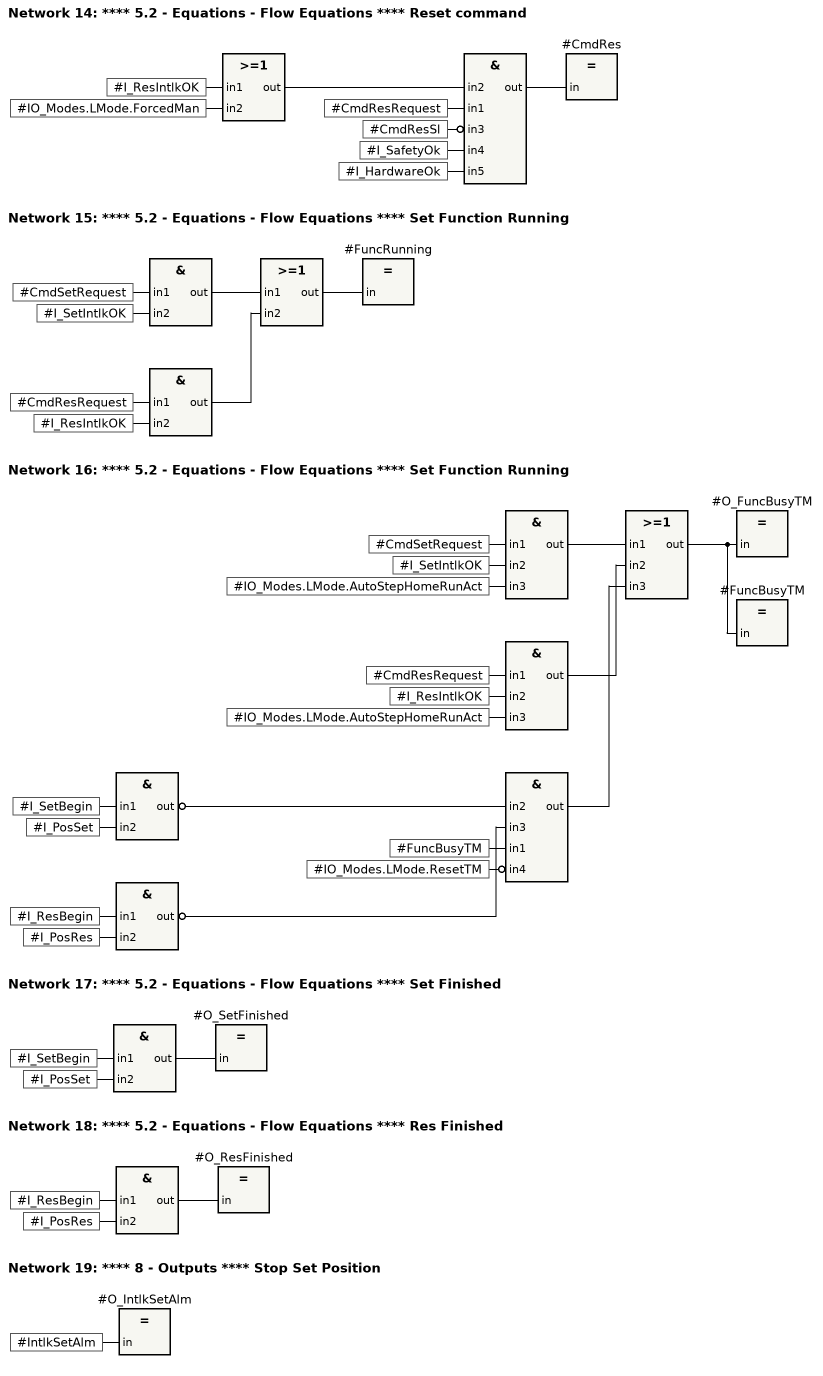
   #CmdRes := (#I_ResIntlkOK OR #IO_Modes.LMode.ForcedMan) AND #CmdResRequest AND NOT #CmdResSl AND #I_SafetyOk AND #I_HardwareOk;
END_REGION

REGION Network 15: **** 5.2 - Equations - Flow Equations **** Set Function Running
   // Set Function Running
   #FuncRunning := (#CmdSetRequest AND #I_SetIntlkOK) OR (#CmdResRequest AND #I_ResIntlkOK);
END_REGION

REGION Network 16: **** 5.2 - Equations - Flow Equations **** Set Function Running
   // Set Function Running
   #O_FuncBusyTM := (#CmdSetRequest AND #I_SetIntlkOK AND #IO_Modes.LMode.AutoStepHomeRunAct) OR (#CmdResRequest AND #I_ResIntlkOK AND #IO_Modes.LMode.AutoStepHomeRunAct) OR (NOT (#I_SetBegin AND #I_PosSet) AND NOT (#I_ResBegin AND #I_PosRes) AND #FuncBusyTM AND NOT #IO_Modes.LMode.ResetTM);
   #FuncBusyTM := #O_FuncBusyTM;
END_REGION

REGION Network 17: **** 5.2 - Equations - Flow Equations **** Set Finished
   // Set Finished
   #O_SetFinished := #I_SetBegin AND #I_PosSet;
END_REGION

REGION Network 18: **** 5.2 - Equations - Flow Equations **** Res Finished
   // Res Finished
   #O_ResFinished := #I_ResBegin AND #I_PosRes;
END_REGION

REGION Network 19: **** 8 - Outputs **** Stop Set Position
   // Stop Set Position
   #O_IntlkSetAlm := #IntlkSetAlm;
END_REGION

REGION Network 20: **** 8 - Outputs **** Stop Reset Position
   // Stop Reset Position
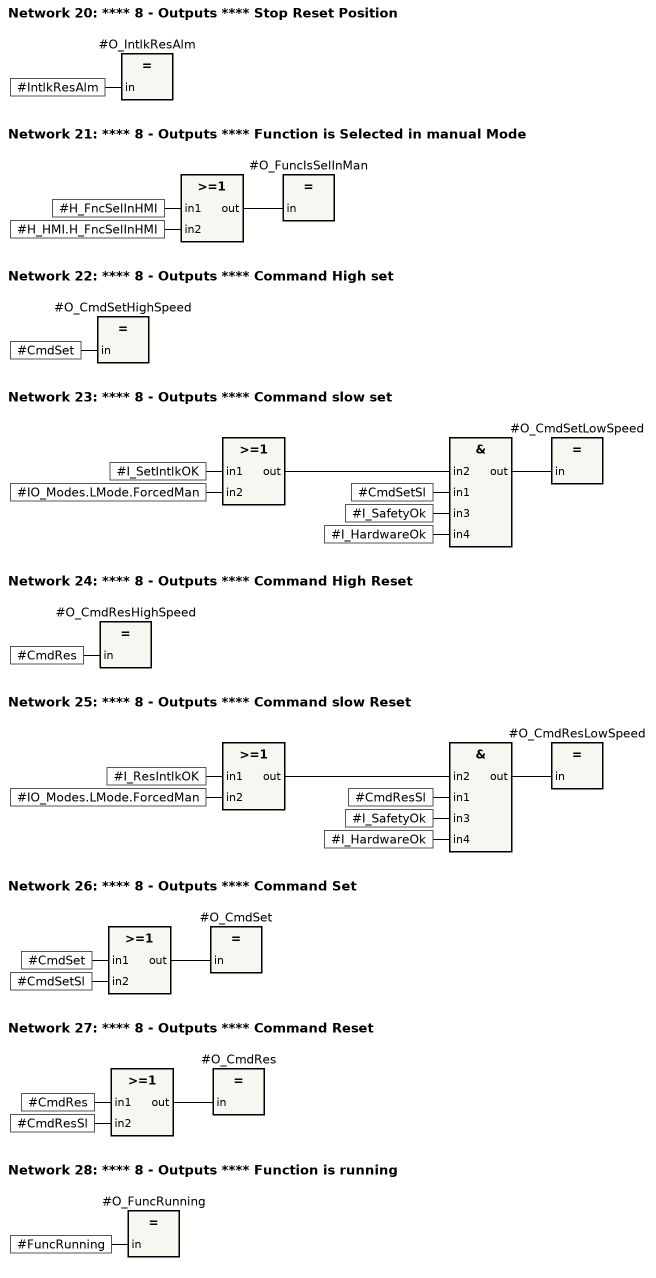
   #O_IntlkResAlm := #IntlkResAlm;
END_REGION

REGION Network 21: **** 8 - Outputs **** Function is Selected in manual Mode
   // Function is Selected in manual Mode
   #O_FuncIsSelInMan := #H_FncSelInHMI OR #H_HMI.H_FncSelInHMI;
END_REGION

REGION Network 22: **** 8 - Outputs **** Command High set
   // Command set
   #O_CmdSetHighSpeed := #CmdSet;
END_REGION

REGION Network 23: **** 8 - Outputs **** Command slow set
   // Command slow set
   #O_CmdSetLowSpeed := (#I_SetIntlkOK OR #IO_Modes.LMode.ForcedMan) AND #CmdSetSl AND #I_SafetyOk AND #I_HardwareOk;
END_REGION

REGION Network 24: **** 8 - Outputs **** Command High Reset
   // Command Reset
   #O_CmdResHighSpeed := #CmdRes;
END_REGION

REGION Network 25: **** 8 - Outputs **** Command slow Reset
   // Command slow Reset
   #O_CmdResLowSpeed := (#I_ResIntlkOK OR #IO_Modes.LMode.ForcedMan) AND #CmdResSl AND #I_SafetyOk AND #I_HardwareOk;
END_REGION

REGION Network 26: **** 8 - Outputs **** Command Set
   // Command set
   #O_CmdSet := #CmdSet OR #CmdSetSl;
END_REGION

REGION Network 27: **** 8 - Outputs **** Command Reset
   // Command Reset
   #O_CmdRes := #CmdRes OR #CmdResSl;
END_REGION

REGION Network 28: **** 8 - Outputs **** Function is running
   // Function is running
   #O_FuncRunning := #FuncRunning;
END_REGION

REGION Network 29: **** 8 - Outputs **** LED - Indication
   // LED - Indication
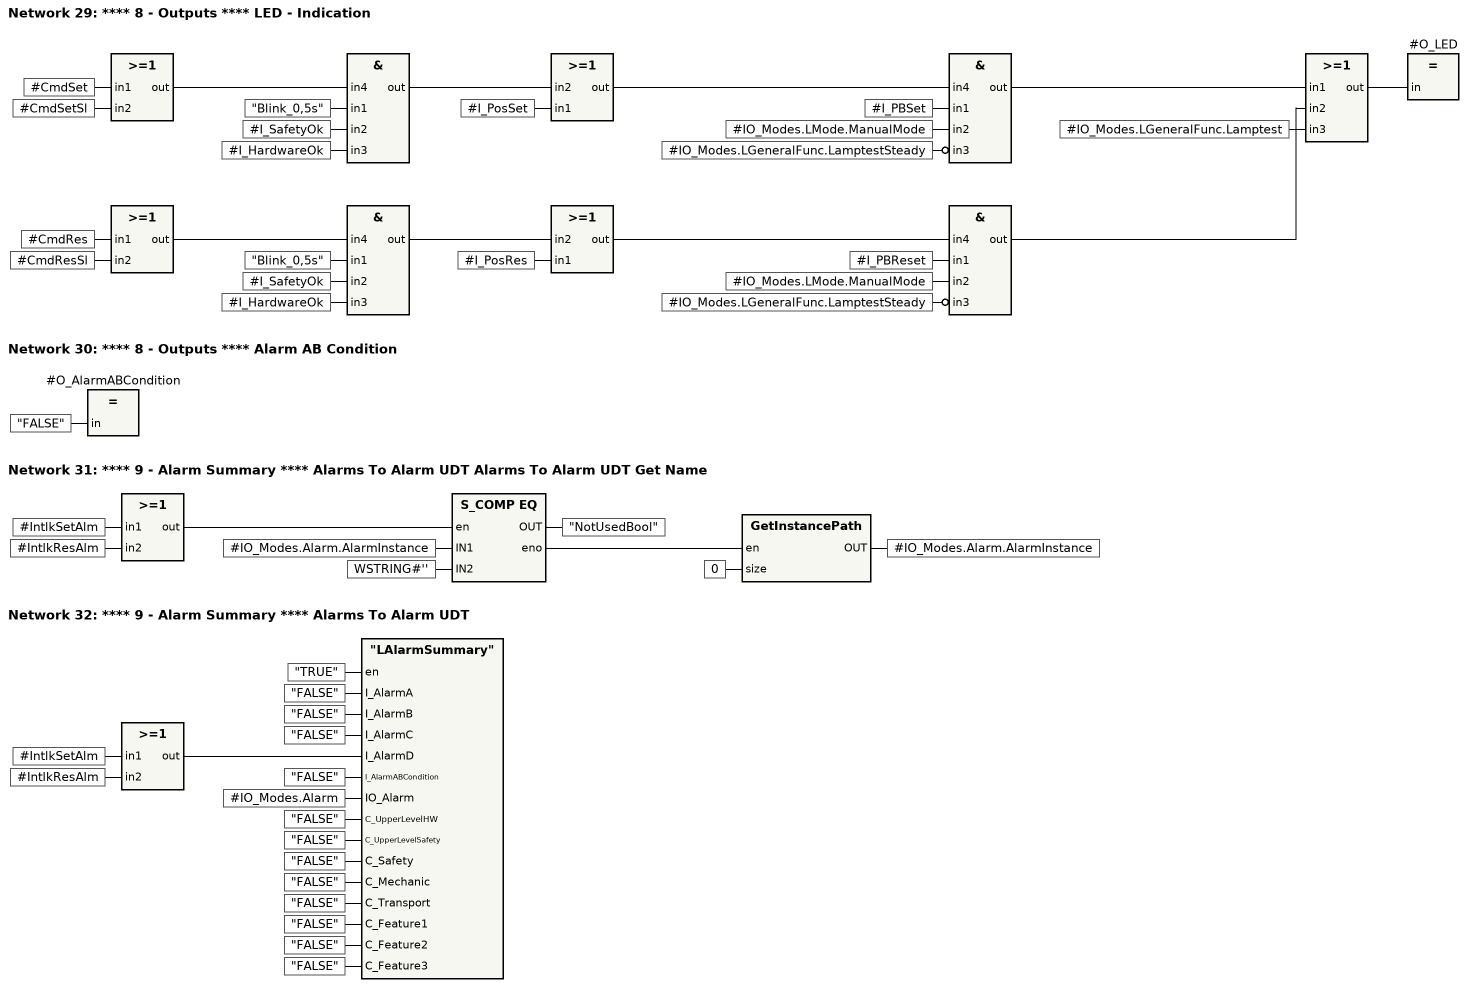
   #O_LED := ((((#CmdSet OR #CmdSetSl) AND "Blink_0,5s" AND #I_SafetyOk AND #I_HardwareOk) OR #I_PosSet) AND #I_PBSet AND #IO_Modes.LMode.ManualMode AND NOT #IO_Modes.LGeneralFunc.LamptestSteady) OR ((((#CmdRes OR #CmdResSl) AND "Blink_0,5s" AND #I_SafetyOk AND #I_HardwareOk) OR #I_PosRes) AND #I_PBReset AND #IO_Modes.LMode.ManualMode AND NOT #IO_Modes.LGeneralFunc.LamptestSteady) OR #IO_Modes.LGeneralFunc.Lamptest;
END_REGION

REGION Network 30: **** 8 - Outputs **** Alarm AB Condition
   // Alarm AB Condition
   #O_AlarmABCondition := "FALSE";
END_REGION

REGION Network 31: **** 9 - Alarm Summary **** Alarms To Alarm UDT Alarms To Alarm UDT Get Name
   // Alarm D
   S_COMP(EN := #IntlkSetAlm OR #IntlkResAlm,
          IN1 := #IO_Modes.Alarm.AlarmInstance,
          IN2 := WSTRING#'',
          OUT => "NotUsedBool",
          ENO => #_w1);
   IF #_w1 THEN GetInstancePath(size := 0, OUT => #IO_Modes.Alarm.AlarmInstance); END_IF;
END_REGION

REGION Network 32: **** 9 - Alarm Summary **** Alarms To Alarm UDT
   // Alarm D
   IF "TRUE" THEN
       "LAlarmSummary"(I_AlarmA := "FALSE",
                       I_AlarmB := "FALSE",
                       I_AlarmC := "FALSE",
                       I_AlarmD := #IntlkSetAlm OR #IntlkResAlm,
                       I_AlarmABCondition := "FALSE",
                       IO_Alarm := #IO_Modes.Alarm,
                       C_UpperLevelHW := "FALSE",
                       C_UpperLevelSafety := "FALSE",
                       C_Safety := "FALSE",
                       C_Mechanic := "FALSE",
                       C_Transport := "FALSE",
                       C_Feature1 := "FALSE",
                       C_Feature2 := "FALSE",
                       C_Feature3 := "FALSE");
   END_IF;
END_REGION
END_FUNCTION_BLOCK

FUNCTION_BLOCK "LMovFnc3Pos"   // FB2187, FBD
TITLE = LMovFnc3Pos
{ S7_Optimized_Access := 'TRUE' }
AUTHOR : VCC
FAMILY : Tooling
VERSION : 0.1
// =============================================================================
// This module will be used for the steering of a three Position movement.
// It will get the commands from different Modes, evaluate the status of the 
// Interlock and give the command to the Actuator or direct to simple outputs.
// =============================================================================
// stored: AutoNumber false, IsIECCheckEnabled false, IsRetainMemResEnabled false, MemoryReserve 100, SetENOAutomatically False, UDAEnableTagReadback false
   VAR_INPUT
      I_Pos1 { ExternalAccessible := 'False'; ExternalVisible := 'False'; ExternalWritable := 'False'} : Bool;   // Position Set detection or summary / Position 1 Detection
      I_Pos2 { ExternalAccessible := 'False'; ExternalVisible := 'False'; ExternalWritable := 'False'} : Bool;   // Position 2 Detection
      I_Pos3 { ExternalAccessible := 'False'; ExternalVisible := 'False'; ExternalWritable := 'False'} : Bool;   // Position Reset detection or summary / Position 3 Detection
      I_PBSet { ExternalAccessible := 'False'; ExternalVisible := 'False'; ExternalWritable := 'False'} : Bool;   // Push button for Set direction (used in manual with button OP panels )
      I_PBReset { ExternalAccessible := 'False'; ExternalVisible := 'False'; ExternalWritable := 'False'} : Bool;   // Push button for reset direcion (used in manual with pushbutton OP panels) / Push button for Reset direction (used in manual with Pushbutton OP panels)
      I_Pos1Begin { ExternalAccessible := 'False'; ExternalVisible := 'False'; ExternalWritable := 'False'} : Bool;   // Function Set begin selection / Function Pos1 begin selection
      I_Pos2Begin { ExternalAccessible := 'False'; ExternalVisible := 'False'; ExternalWritable := 'False'} : Bool;   // Function Set begin selection / Function Pos2 begin selection
      I_Pos3Begin { ExternalAccessible := 'False'; ExternalVisible := 'False'; ExternalWritable := 'False'} : Bool;   // Function Reset begin selection / Function Pos3 begin selection
      I_Pos1IntlkOK { ExternalAccessible := 'False'; ExternalVisible := 'False'; ExternalWritable := 'False'} : Bool;   // Set Interlock / Pos1 Interlock
      I_Pos2IntlkOK { ExternalAccessible := 'False'; ExternalVisible := 'False'; ExternalWritable := 'False'} : Bool;   // Set Interlock / Pos2 Interlock
      I_Pos3IntlkOK { ExternalAccessible := 'False'; ExternalVisible := 'False'; ExternalWritable := 'False'} : Bool;   // Reset Interlock / Pos3 Interlock
      I_MiddleReachedManSTOP { ExternalAccessible := 'False'; ExternalVisible := 'False'; ExternalWritable := 'False'} : Bool;   // Middle pos reached
      I_SafetyOk { ExternalAccessible := 'False'; ExternalVisible := 'False'; ExternalWritable := 'False'} : Bool;   // Safety Ok
      I_HardwareOk { ExternalAccessible := 'False'; ExternalVisible := 'False'; ExternalWritable := 'False'} : Bool;   // Safety Ok / Hardware Ok
   END_VAR
   VAR_OUTPUT
      O_CmdPos1 { ExternalAccessible := 'False'; ExternalVisible := 'False'; ExternalWritable := 'False'} : Bool;   // Command to activate Set movement / Command to Activate Pos1 movement
      O_CmdPos2 { ExternalAccessible := 'False'; ExternalVisible := 'False'; ExternalWritable := 'False'} : Bool;   // Command to activate Set movement / Command to Activate Pos2 movement
      O_CmdPos3 { ExternalAccessible := 'False'; ExternalVisible := 'False'; ExternalWritable := 'False'} : Bool;   // Command to activate Reset movement / Command to Activate Pos3 movement
      O_FuncRunning { ExternalAccessible := 'False'; ExternalVisible := 'False'; ExternalWritable := 'False'} : Bool;   // Signal that the function is running
      O_FuncBusyTM { ExternalAccessible := 'False'; ExternalVisible := 'False'; ExternalWritable := 'False'} : Bool;   // Memory Signal that the function is busy
      O_Pos1Finished { ExternalAccessible := 'False'; ExternalVisible := 'False'; ExternalWritable := 'False'} : Bool;   // Function Set finished to Master Sequencing / Function Pos1 finished to Master Sequencing
      O_Pos2Finished { ExternalAccessible := 'False'; ExternalVisible := 'False'; ExternalWritable := 'False'} : Bool;   // Function Set finished to Master Sequencing / Function Pos2 finished to Master Sequencing
      O_Pos3Finished { ExternalAccessible := 'False'; ExternalVisible := 'False'; ExternalWritable := 'False'} : Bool;   // Function Reset finished to Master Sequencing / Function Pos3 finished to Master Sequencing
      O_IntlkPos1Alm { ExternalAccessible := 'False'; ExternalVisible := 'False'; ExternalWritable := 'False'} : Bool;   // Alarm interlock Set / Alarm Interlock Pos1
      O_IntlkPos2Alm { ExternalAccessible := 'False'; ExternalVisible := 'False'; ExternalWritable := 'False'} : Bool;   // Alarm interlock Set / Alarm Interlock Pos2
      O_IntlkPos3Alm { ExternalAccessible := 'False'; ExternalVisible := 'False'; ExternalWritable := 'False'} : Bool;   // Alarm interlock Reset / Alarm Interlock Reset
      O_FuncIsSelInMan { ExternalAccessible := 'False'; ExternalVisible := 'False'; ExternalWritable := 'False'} : Bool;   // The function is selected in manual mode / The function is Selected in manual Mode
      O_LED { ExternalAccessible := 'False'; ExternalVisible := 'False'; ExternalWritable := 'False'} : Bool;   // LED - Indication
      O_AlarmABCondition { ExternalAccessible := 'False'; ExternalVisible := 'False'; ExternalWritable := 'False'} : Bool;   // Alarms AB condition / Alarm AB Condition
   END_VAR
   VAR_IN_OUT
      IO_Modes : "Modes";   // Modes
      H_HMI : "H_HMI";   // Animation
      H_MovFnc3Pos : "H_MovFnc3Pos";   // Animation
      H_FncSelInHMI { ExternalAccessible := 'False'; ExternalVisible := 'False'; ExternalWritable := 'False'} : Bool;   // This function is selected to run from HMI / This function is Selected to run from HMI
      C_AlarmResetUsed { ExternalAccessible := 'False'; ExternalVisible := 'False'; ExternalWritable := 'False'} : Bool;   // If true, the alrms will be stored untill reseted / If TRUE The Alarms will be stored untill Reseted
      C_EnableMemBegin { ExternalAccessible := 'False'; ExternalVisible := 'False'; ExternalWritable := 'False'} : Bool;   // Enable memory Begin (Command request is memorised until pos reached) / Enable memory Begin (Command Request is memorised until pos reached)
      C_EnIntlkAlm { ExternalAccessible := 'False'; ExternalVisible := 'False'; ExternalWritable := 'False'} : Bool := TRUE;   // Enable Interlock Alarm
      C_SetReset { ExternalAccessible := 'False'; ExternalVisible := 'False'; ExternalWritable := 'False'} : Bool;   // Enable Set Reset Functionality ( If enabled output is kept until the Cmd direction is changed )
      C_ForceManual { ExternalAccessible := 'False'; ExternalVisible := 'False'; ExternalWritable := 'False'} : Bool := FALSE;   // Force Manual
   END_VAR
   VAR
      ResetAlarm { ExternalAccessible := 'False'; ExternalVisible := 'False'; ExternalWritable := 'False'} : Bool;   // Reset Alarm Memory
      CmdPos1Request { ExternalAccessible := 'False'; ExternalVisible := 'False'; ExternalWritable := 'False'} : Bool;   // Set Command request to activate the interlock / Pos1 Command Request to Activate the Interlock
      CmdPos2Request { ExternalAccessible := 'False'; ExternalVisible := 'False'; ExternalWritable := 'False'} : Bool;   // Set Command request to activate the interlock / Pos1 Command Request to Activate the Interlock
      CmdPos3Request { ExternalAccessible := 'False'; ExternalVisible := 'False'; ExternalWritable := 'False'} : Bool;   // Reset Command request to activate the interlock / Pos3 Command Request to Activate the Interlock
      EdgeStopDetPos1 { ExternalAccessible := 'False'; ExternalVisible := 'False'; ExternalWritable := 'False'} : Bool;   // Edge on stop detection to be abble to go over it in force manual
      EdgeStopDetPos2 { ExternalAccessible := 'False'; ExternalVisible := 'False'; ExternalWritable := 'False'} : Bool;   // Edge on stop detection to be abble to go over it in force manual
      EdgeStopDetPos3 { ExternalAccessible := 'False'; ExternalVisible := 'False'; ExternalWritable := 'False'} : Bool;   // Edge on stop detection to be abble to go over it in force manual
      IntlkPos1Alm { ExternalAccessible := 'False'; ExternalVisible := 'False'; ExternalWritable := 'False'} : Bool;   // Alarm interlock Set / Alarm Interlock Pos1
      IntlkPos2Alm { ExternalAccessible := 'False'; ExternalVisible := 'False'; ExternalWritable := 'False'} : Bool;   // Alarm interlock Set / Alarm Interlock Pos2
      IntlkPos3Alm { ExternalAccessible := 'False'; ExternalVisible := 'False'; ExternalWritable := 'False'} : Bool;   // Alarm interlock Reset / Alarm Interlock Reset
      CmdPos1 { ExternalAccessible := 'False'; ExternalVisible := 'False'; ExternalWritable := 'False'} : Bool;   // Command to activate Set movement / Command to Activate Pos1 movement
      CmdPos2 { ExternalAccessible := 'False'; ExternalVisible := 'False'; ExternalWritable := 'False'} : Bool;   // Command to activate Set movement / Command to Activate Pos2 movement
      CmdPos3 { ExternalAccessible := 'False'; ExternalVisible := 'False'; ExternalWritable := 'False'} : Bool;   // Command to activate Reset movement / Command to Activate Pos3 movement
      IntlkPos1AlmCond { ExternalAccessible := 'False'; ExternalVisible := 'False'; ExternalWritable := 'False'} : Bool;   // Alarm interlock Set condition / Alarm Interlock Pos1 condition
      IntlkPos2AlmCond { ExternalAccessible := 'False'; ExternalVisible := 'False'; ExternalWritable := 'False'} : Bool;   // Alarm interlock Set condition / Alarm Interlock Pos2 condition
      IntlkPos3AlmCond { ExternalAccessible := 'False'; ExternalVisible := 'False'; ExternalWritable := 'False'} : Bool;   // Alarm interlock Reset condition / Alarm Interlock Pos3 condition
      FuncRunning { ExternalAccessible := 'False'; ExternalVisible := 'False'; ExternalWritable := 'False'} : Bool;   // Function is running
      LampTest { ExternalAccessible := 'False'; ExternalVisible := 'False'; ExternalWritable := 'False'} : Bool;   // Lamp test
      LampTestSteady { ExternalAccessible := 'False'; ExternalVisible := 'False'; ExternalWritable := 'False'} : Bool;   // Lamp test always on from mode of station / Lamp test always on from Mode of station
      FuncBusyTM { ExternalAccessible := 'False'; ExternalVisible := 'False'; ExternalWritable := 'False'} : Bool;   // Memory Signal that the function is busy
      AlarmTimer { ExternalAccessible := 'False'; ExternalVisible := 'False'; ExternalWritable := 'False'} : "LTimer";
      AlmFilterResult { ExternalAccessible := 'False'; ExternalVisible := 'False'; ExternalWritable := 'False'} : Bool;
   END_VAR
   VAR_TEMP   // added for the SCL form of the ladder/FBD networks
      _w1 : Bool;
   END_VAR
BEGIN

REGION Network 1: **** 2.2 - Alarms - Alarm Generation **** Alarm Filter
   // Alarm Filter
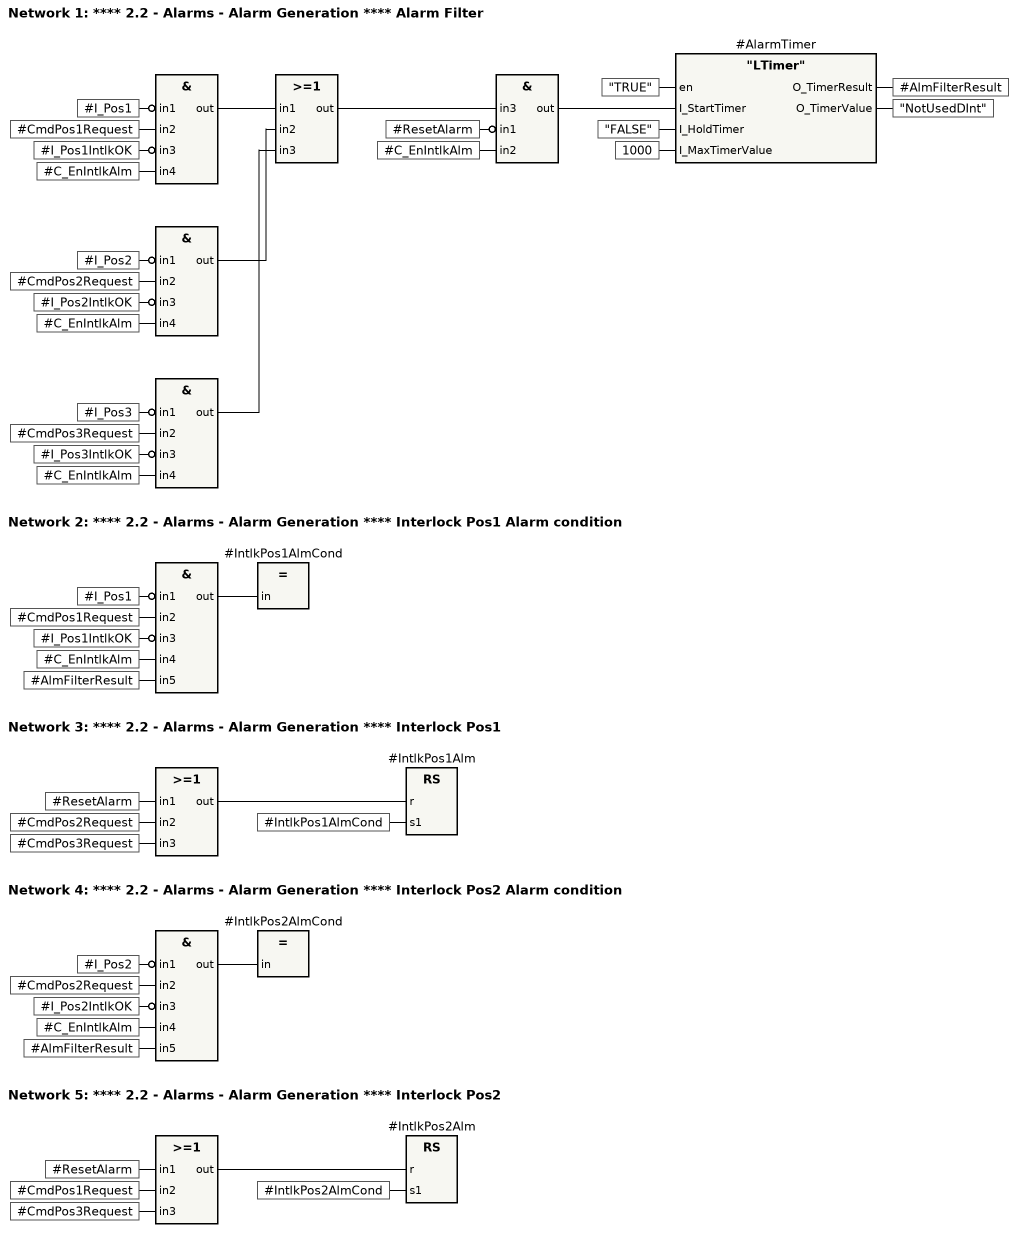
   IF "TRUE" THEN
       #AlarmTimer(I_StartTimer := ((NOT #I_Pos1 AND #CmdPos1Request AND NOT #I_Pos1IntlkOK AND #C_EnIntlkAlm) OR (NOT #I_Pos2 AND #CmdPos2Request AND NOT #I_Pos2IntlkOK AND #C_EnIntlkAlm) OR (NOT #I_Pos3 AND #CmdPos3Request AND NOT #I_Pos3IntlkOK AND #C_EnIntlkAlm)) AND NOT #ResetAlarm AND #C_EnIntlkAlm,   // "LTimer"
                   I_HoldTimer := "FALSE",
                   I_MaxTimerValue := 1000,
                   O_TimerResult => #AlmFilterResult,
                   O_TimerValue => "NotUsedDInt");
   END_IF;
END_REGION

REGION Network 2: **** 2.2 - Alarms - Alarm Generation **** Interlock Pos1 Alarm condition
   // Interlock Pos1 Alarm condition
   #IntlkPos1AlmCond := NOT #I_Pos1 AND #CmdPos1Request AND NOT #I_Pos1IntlkOK AND #C_EnIntlkAlm AND #AlmFilterResult;
END_REGION

REGION Network 3: **** 2.2 - Alarms - Alarm Generation **** Interlock Pos1
   // Interlock Pos1
   IF #ResetAlarm OR #CmdPos2Request OR #CmdPos3Request THEN
       #IntlkPos1Alm := FALSE;   // RS flip-flop
   END_IF;
   IF #IntlkPos1AlmCond THEN #IntlkPos1Alm := TRUE; END_IF;
END_REGION

REGION Network 4: **** 2.2 - Alarms - Alarm Generation **** Interlock Pos2 Alarm condition
   // Interlock Pos2 Alarm condition
   #IntlkPos2AlmCond := NOT #I_Pos2 AND #CmdPos2Request AND NOT #I_Pos2IntlkOK AND #C_EnIntlkAlm AND #AlmFilterResult;
END_REGION

REGION Network 5: **** 2.2 - Alarms - Alarm Generation **** Interlock Pos2
   // Interlock Pos2
   IF #ResetAlarm OR #CmdPos1Request OR #CmdPos3Request THEN
       #IntlkPos2Alm := FALSE;   // RS flip-flop
   END_IF;
   IF #IntlkPos2AlmCond THEN #IntlkPos2Alm := TRUE; END_IF;
END_REGION

REGION Network 6: **** 2.2 - Alarms - Alarm Generation **** Interlock Pos3 Alarm condition
   // Interlock Pos3 Alarm condition
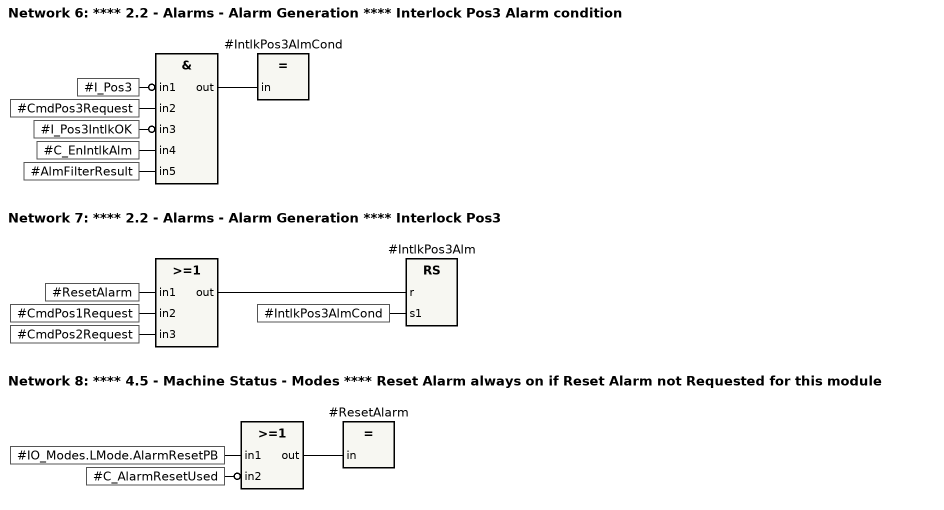
   #IntlkPos3AlmCond := NOT #I_Pos3 AND #CmdPos3Request AND NOT #I_Pos3IntlkOK AND #C_EnIntlkAlm AND #AlmFilterResult;
END_REGION

REGION Network 7: **** 2.2 - Alarms - Alarm Generation **** Interlock Pos3
   // Interlock Pos3
   IF #ResetAlarm OR #CmdPos1Request OR #CmdPos2Request THEN
       #IntlkPos3Alm := FALSE;   // RS flip-flop
   END_IF;
   IF #IntlkPos3AlmCond THEN #IntlkPos3Alm := TRUE; END_IF;
END_REGION

REGION Network 8: **** 4.5 - Machine Status - Modes **** Reset Alarm always on if Reset Alarm not Requested for this module
   // Reset Alarm always on if Reset Alarm not Requested for this module
   #ResetAlarm := #IO_Modes.LMode.AlarmResetPB OR NOT #C_AlarmResetUsed;
END_REGION

REGION Network 9: **** 4.6 - Machine Status - Indication **** Icon Animation
   // Icon Animation
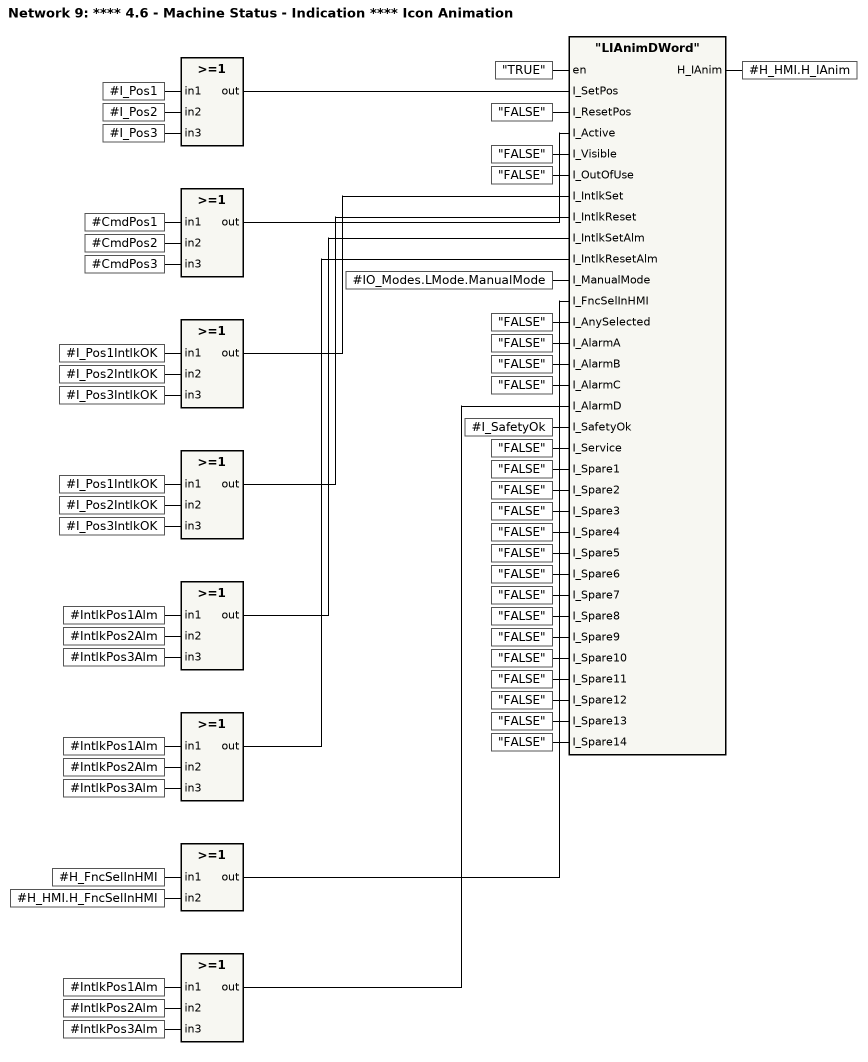
   IF "TRUE" THEN
       "LIAnimDWord"(I_SetPos := #I_Pos1 OR #I_Pos2 OR #I_Pos3,
                     I_ResetPos := "FALSE",
                     I_Active := #CmdPos1 OR #CmdPos2 OR #CmdPos3,
                     I_Visible := "FALSE",
                     I_OutOfUse := "FALSE",
                     I_IntlkSet := #I_Pos1IntlkOK OR #I_Pos2IntlkOK OR #I_Pos3IntlkOK,
                     I_IntlkReset := #I_Pos1IntlkOK OR #I_Pos2IntlkOK OR #I_Pos3IntlkOK,
                     I_IntlkSetAlm := #IntlkPos1Alm OR #IntlkPos2Alm OR #IntlkPos3Alm,
                     I_IntlkResetAlm := #IntlkPos1Alm OR #IntlkPos2Alm OR #IntlkPos3Alm,
                     I_ManualMode := #IO_Modes.LMode.ManualMode,
                     I_FncSelInHMI := #H_FncSelInHMI OR #H_HMI.H_FncSelInHMI,
                     I_AnySelected := "FALSE",
                     I_AlarmA := "FALSE",
                     I_AlarmB := "FALSE",
                     I_AlarmC := "FALSE",
                     I_AlarmD := #IntlkPos1Alm OR #IntlkPos2Alm OR #IntlkPos3Alm,
                     I_SafetyOk := #I_SafetyOk,
                     I_Service := "FALSE",
                     I_Spare1 := "FALSE",
                     I_Spare2 := "FALSE",
                     I_Spare3 := "FALSE",
                     I_Spare4 := "FALSE",
                     I_Spare5 := "FALSE",
                     I_Spare6 := "FALSE",
                     I_Spare7 := "FALSE",
                     I_Spare8 := "FALSE",
                     I_Spare9 := "FALSE",
                     I_Spare10 := "FALSE",
                     I_Spare11 := "FALSE",
                     I_Spare12 := "FALSE",
                     I_Spare13 := "FALSE",
                     I_Spare14 := "FALSE",
                     H_IAnim => #H_HMI.H_IAnim);
   END_IF;
END_REGION

REGION Network 10: **** 4.6 - Machine Status - Indication **** Animation
   // Animation
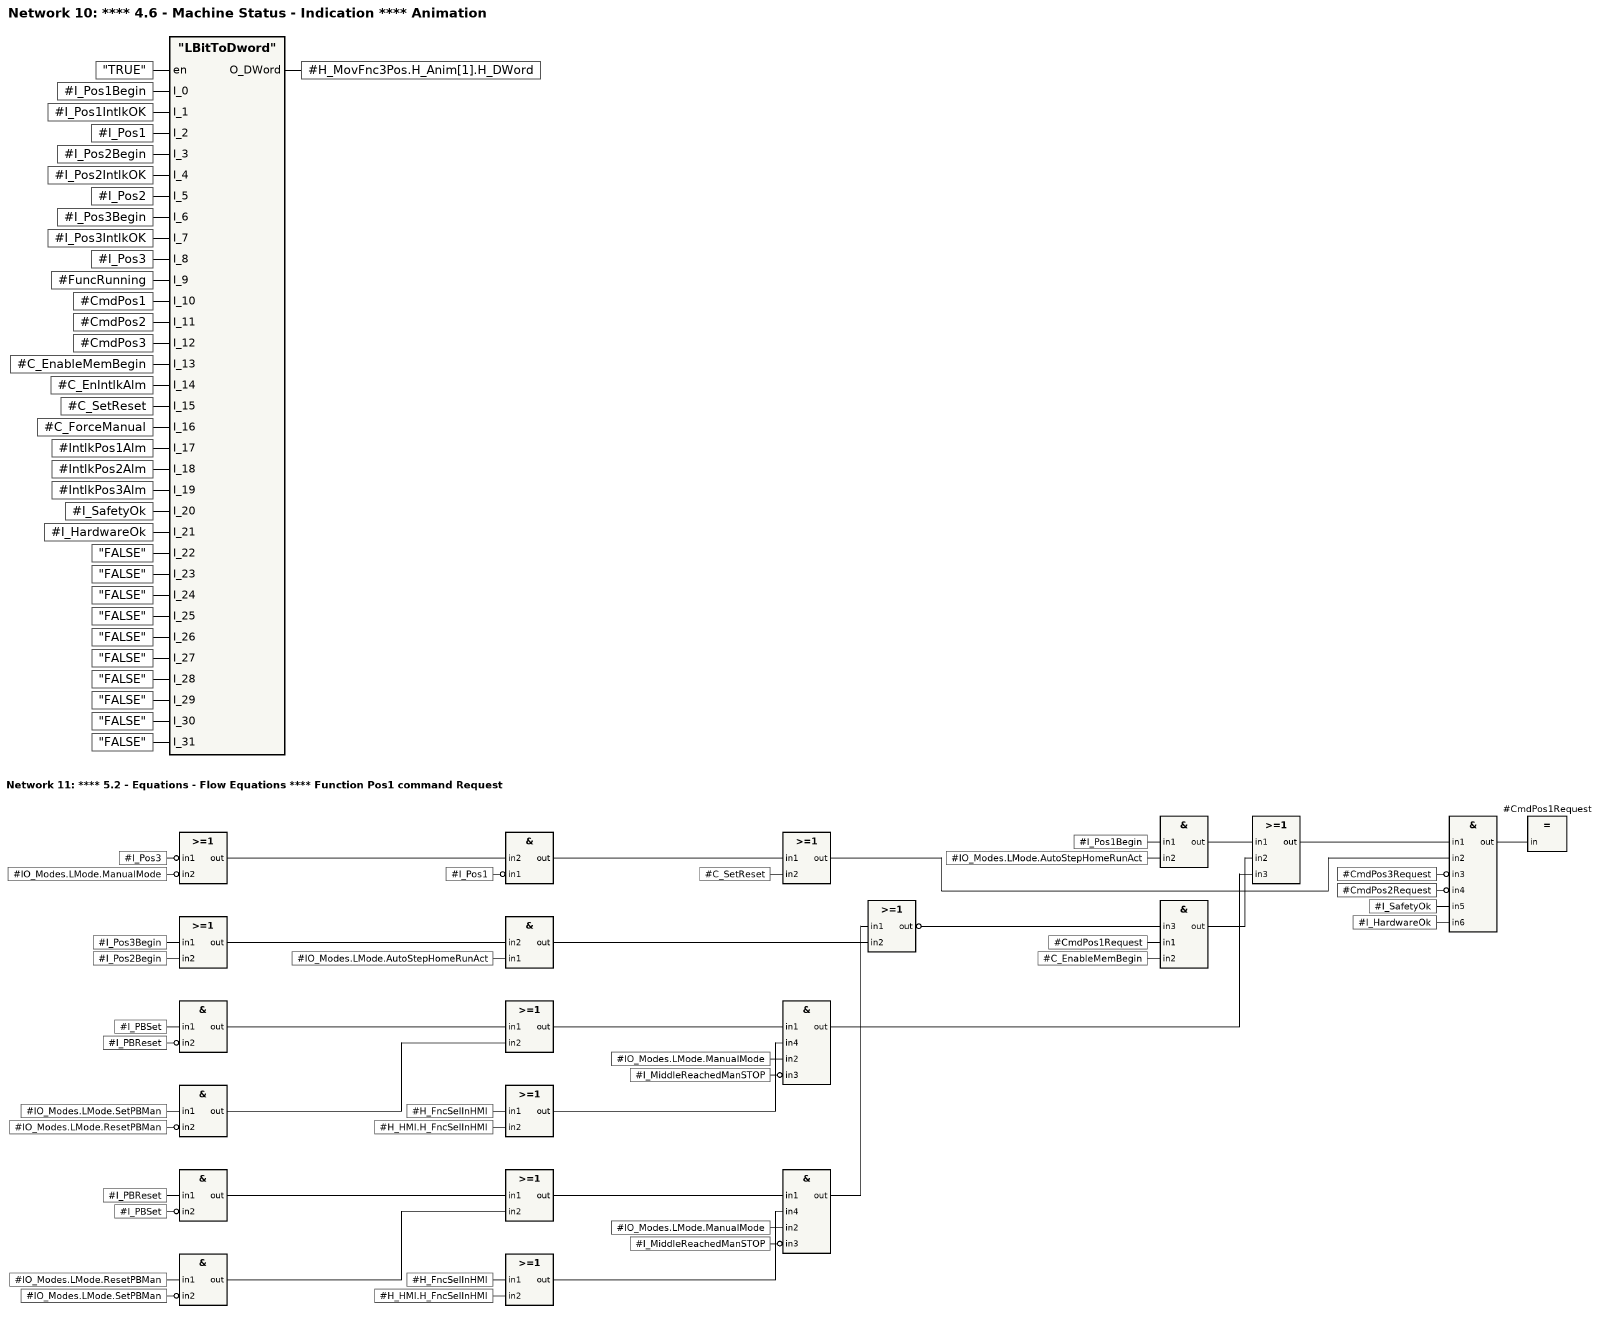
   IF "TRUE" THEN
       "LBitToDword"(I_0 := #I_Pos1Begin,
                     I_1 := #I_Pos1IntlkOK,
                     I_2 := #I_Pos1,
                     I_3 := #I_Pos2Begin,
                     I_4 := #I_Pos2IntlkOK,
                     I_5 := #I_Pos2,
                     I_6 := #I_Pos3Begin,
                     I_7 := #I_Pos3IntlkOK,
                     I_8 := #I_Pos3,
                     I_9 := #FuncRunning,
                     I_10 := #CmdPos1,
                     I_11 := #CmdPos2,
                     I_12 := #CmdPos3,
                     I_13 := #C_EnableMemBegin,
                     I_14 := #C_EnIntlkAlm,
                     I_15 := #C_SetReset,
                     I_16 := #C_ForceManual,
                     I_17 := #IntlkPos1Alm,
                     I_18 := #IntlkPos2Alm,
                     I_19 := #IntlkPos3Alm,
                     I_20 := #I_SafetyOk,
                     I_21 := #I_HardwareOk,
                     I_22 := "FALSE",
                     I_23 := "FALSE",
                     I_24 := "FALSE",
                     I_25 := "FALSE",
                     I_26 := "FALSE",
                     I_27 := "FALSE",
                     I_28 := "FALSE",
                     I_29 := "FALSE",
                     I_30 := "FALSE",
                     I_31 := "FALSE",
                     O_DWord => #H_MovFnc3Pos.H_Anim[1].H_DWord);
   END_IF;
END_REGION

REGION Network 11: **** 5.2 - Equations - Flow Equations **** Function Pos1 command Request
   // Function Pos1 command Request
   #CmdPos1Request := ((#I_Pos1Begin AND #IO_Modes.LMode.AutoStepHomeRunAct) OR (NOT ((((#I_PBReset AND NOT #I_PBSet) OR (#IO_Modes.LMode.ResetPBMan AND NOT #IO_Modes.LMode.SetPBMan)) AND (#H_FncSelInHMI OR #H_HMI.H_FncSelInHMI) AND #IO_Modes.LMode.ManualMode AND NOT #I_MiddleReachedManSTOP) OR ((#I_Pos3Begin OR #I_Pos2Begin) AND #IO_Modes.LMode.AutoStepHomeRunAct)) AND #CmdPos1Request AND #C_EnableMemBegin) OR (((#I_PBSet AND NOT #I_PBReset) OR (#IO_Modes.LMode.SetPBMan AND NOT #IO_Modes.LMode.ResetPBMan)) AND (#H_FncSelInHMI OR #H_HMI.H_FncSelInHMI) AND #IO_Modes.LMode.ManualMode AND NOT #I_MiddleReachedManSTOP)) AND (((NOT #I_Pos3 OR NOT #IO_Modes.LMode.ManualMode) AND NOT #I_Pos1) OR #C_SetReset) AND NOT #CmdPos3Request AND NOT #CmdPos2Request AND #I_SafetyOk AND #I_HardwareOk;
END_REGION

REGION Network 12: **** 5.2 - Equations - Flow Equations **** Function Pos2 command Request
   // Function Pos2 command Request
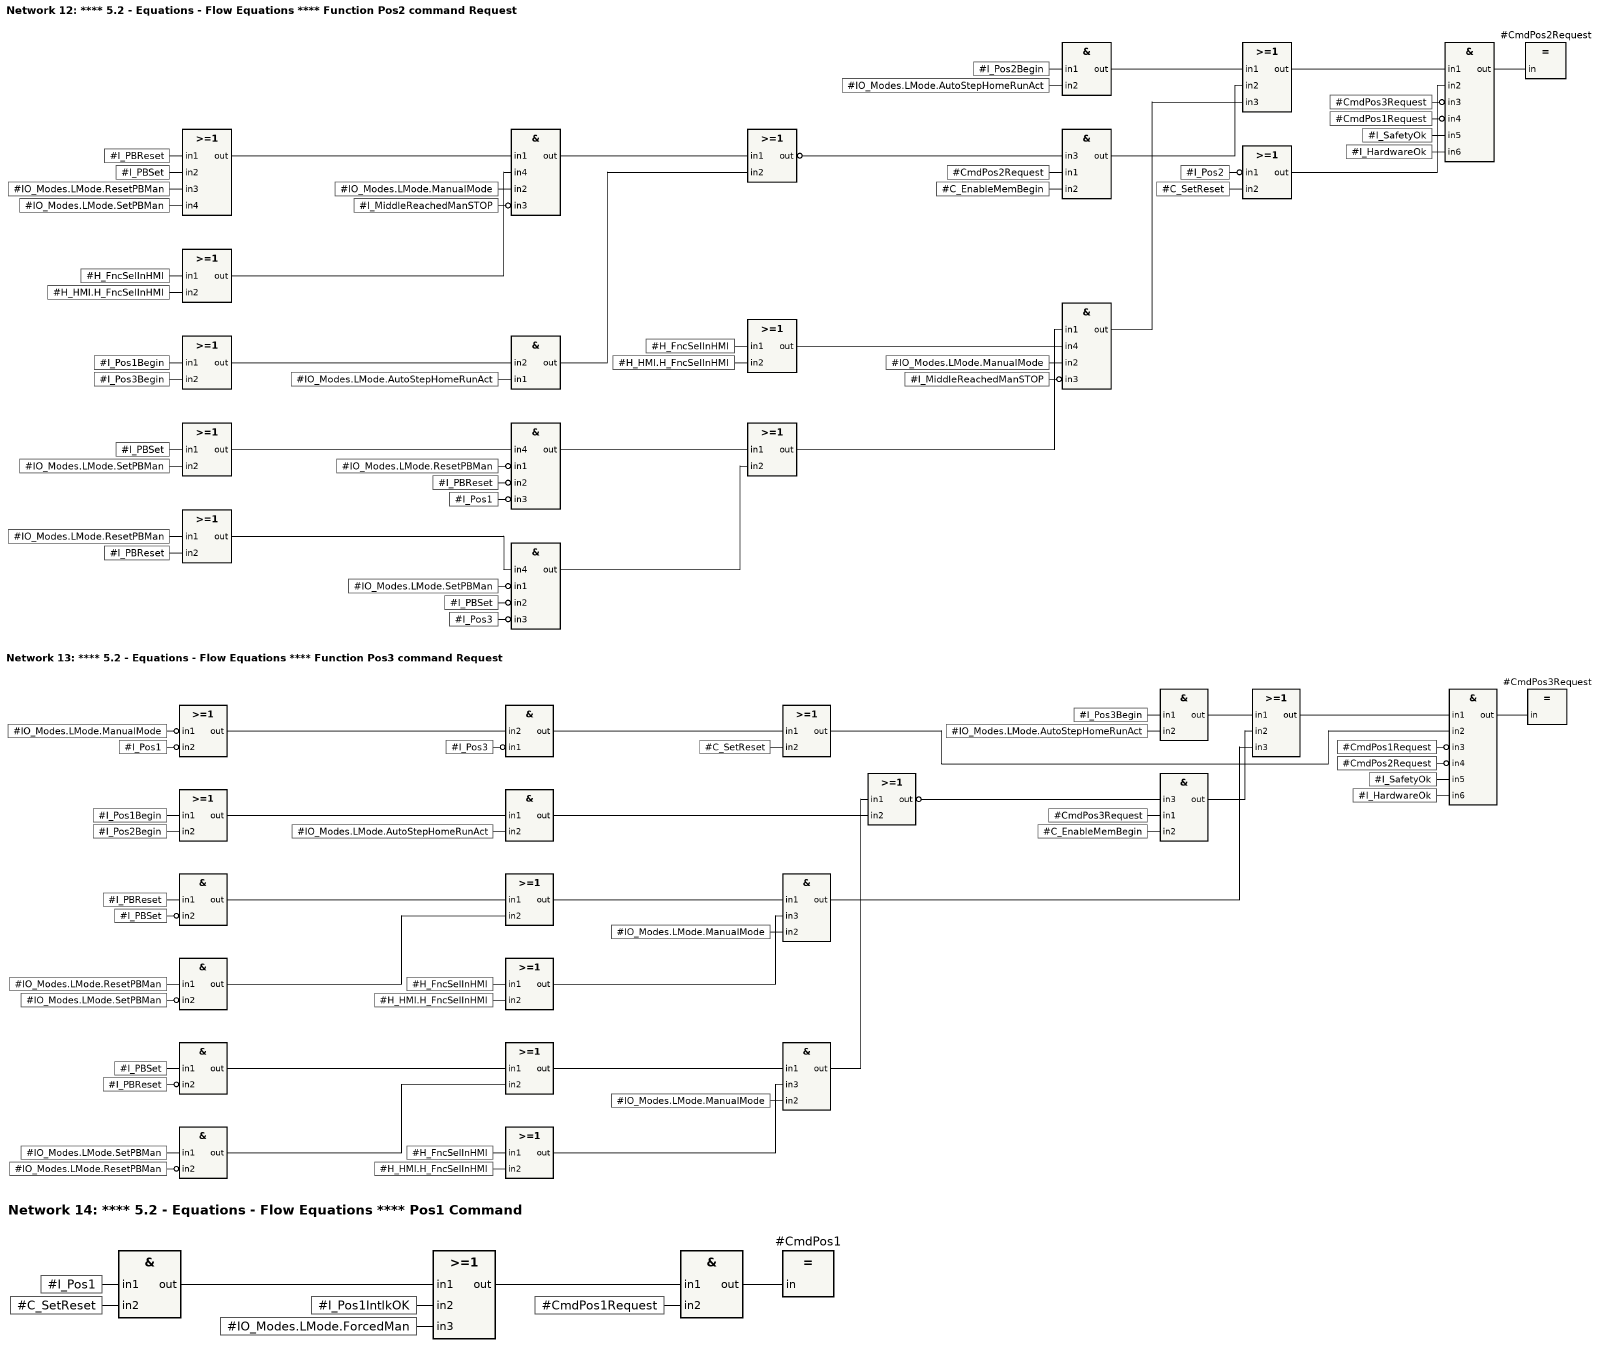
   #CmdPos2Request := ((#I_Pos2Begin AND #IO_Modes.LMode.AutoStepHomeRunAct) OR (NOT (((#I_PBReset OR #I_PBSet OR #IO_Modes.LMode.ResetPBMan OR #IO_Modes.LMode.SetPBMan) AND (#H_FncSelInHMI OR #H_HMI.H_FncSelInHMI) AND #IO_Modes.LMode.ManualMode AND NOT #I_MiddleReachedManSTOP) OR ((#I_Pos1Begin OR #I_Pos3Begin) AND #IO_Modes.LMode.AutoStepHomeRunAct)) AND #CmdPos2Request AND #C_EnableMemBegin) OR ((((#I_PBSet OR #IO_Modes.LMode.SetPBMan) AND NOT #IO_Modes.LMode.ResetPBMan AND NOT #I_PBReset AND NOT #I_Pos1) OR ((#IO_Modes.LMode.ResetPBMan OR #I_PBReset) AND NOT #IO_Modes.LMode.SetPBMan AND NOT #I_PBSet AND NOT #I_Pos3)) AND (#H_FncSelInHMI OR #H_HMI.H_FncSelInHMI) AND #IO_Modes.LMode.ManualMode AND NOT #I_MiddleReachedManSTOP)) AND (NOT #I_Pos2 OR #C_SetReset) AND NOT #CmdPos3Request AND NOT #CmdPos1Request AND #I_SafetyOk AND #I_HardwareOk;
END_REGION

REGION Network 13: **** 5.2 - Equations - Flow Equations **** Function Pos3 command Request
   // Function Pos3 command Request
   #CmdPos3Request := ((#I_Pos3Begin AND #IO_Modes.LMode.AutoStepHomeRunAct) OR (NOT ((((#I_PBSet AND NOT #I_PBReset) OR (#IO_Modes.LMode.SetPBMan AND NOT #IO_Modes.LMode.ResetPBMan)) AND (#H_FncSelInHMI OR #H_HMI.H_FncSelInHMI) AND #IO_Modes.LMode.ManualMode) OR ((#I_Pos1Begin OR #I_Pos2Begin) AND #IO_Modes.LMode.AutoStepHomeRunAct)) AND #CmdPos3Request AND #C_EnableMemBegin) OR (((#I_PBReset AND NOT #I_PBSet) OR (#IO_Modes.LMode.ResetPBMan AND NOT #IO_Modes.LMode.SetPBMan)) AND (#H_FncSelInHMI OR #H_HMI.H_FncSelInHMI) AND #IO_Modes.LMode.ManualMode)) AND (((NOT #IO_Modes.LMode.ManualMode OR NOT #I_Pos1) AND NOT #I_Pos3) OR #C_SetReset) AND NOT #CmdPos1Request AND NOT #CmdPos2Request AND #I_SafetyOk AND #I_HardwareOk;
END_REGION

REGION Network 14: **** 5.2 - Equations - Flow Equations **** Pos1 Command
   // Pos1 Command
   #CmdPos1 := ((#I_Pos1 AND #C_SetReset) OR #I_Pos1IntlkOK OR #IO_Modes.LMode.ForcedMan) AND #CmdPos1Request;
END_REGION

REGION Network 15: **** 5.2 - Equations - Flow Equations **** Pos2 Command
   // Pos2 Command
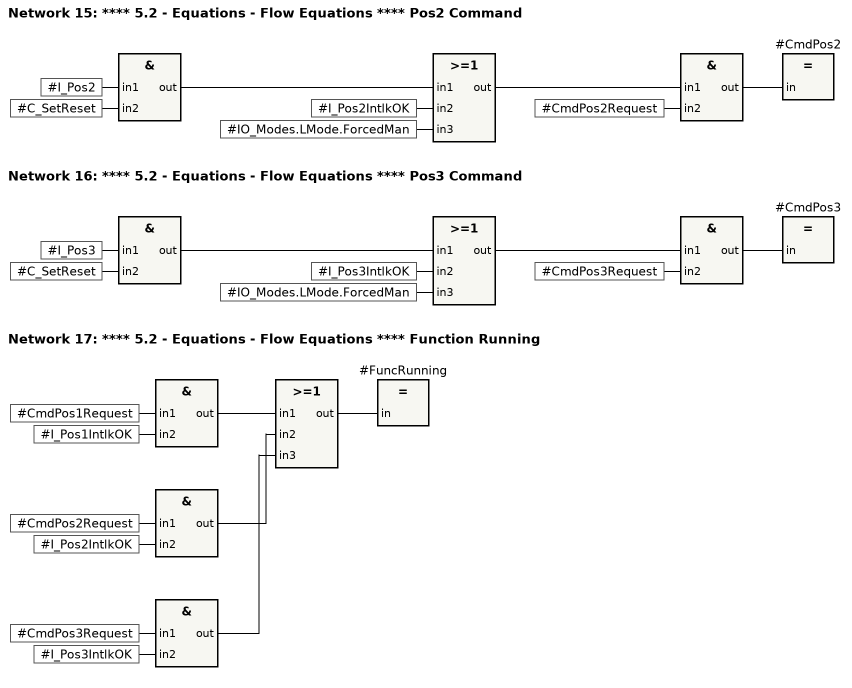
   #CmdPos2 := ((#I_Pos2 AND #C_SetReset) OR #I_Pos2IntlkOK OR #IO_Modes.LMode.ForcedMan) AND #CmdPos2Request;
END_REGION

REGION Network 16: **** 5.2 - Equations - Flow Equations **** Pos3 Command
   // Pos3 Command
   #CmdPos3 := ((#I_Pos3 AND #C_SetReset) OR #I_Pos3IntlkOK OR #IO_Modes.LMode.ForcedMan) AND #CmdPos3Request;
END_REGION

REGION Network 17: **** 5.2 - Equations - Flow Equations **** Function Running
   // Function Running
   #FuncRunning := (#CmdPos1Request AND #I_Pos1IntlkOK) OR (#CmdPos2Request AND #I_Pos2IntlkOK) OR (#CmdPos3Request AND #I_Pos3IntlkOK);
END_REGION

REGION Network 18: **** 5.2 - Equations - Flow Equations **** Function Running Memory
   // Function Running Memory
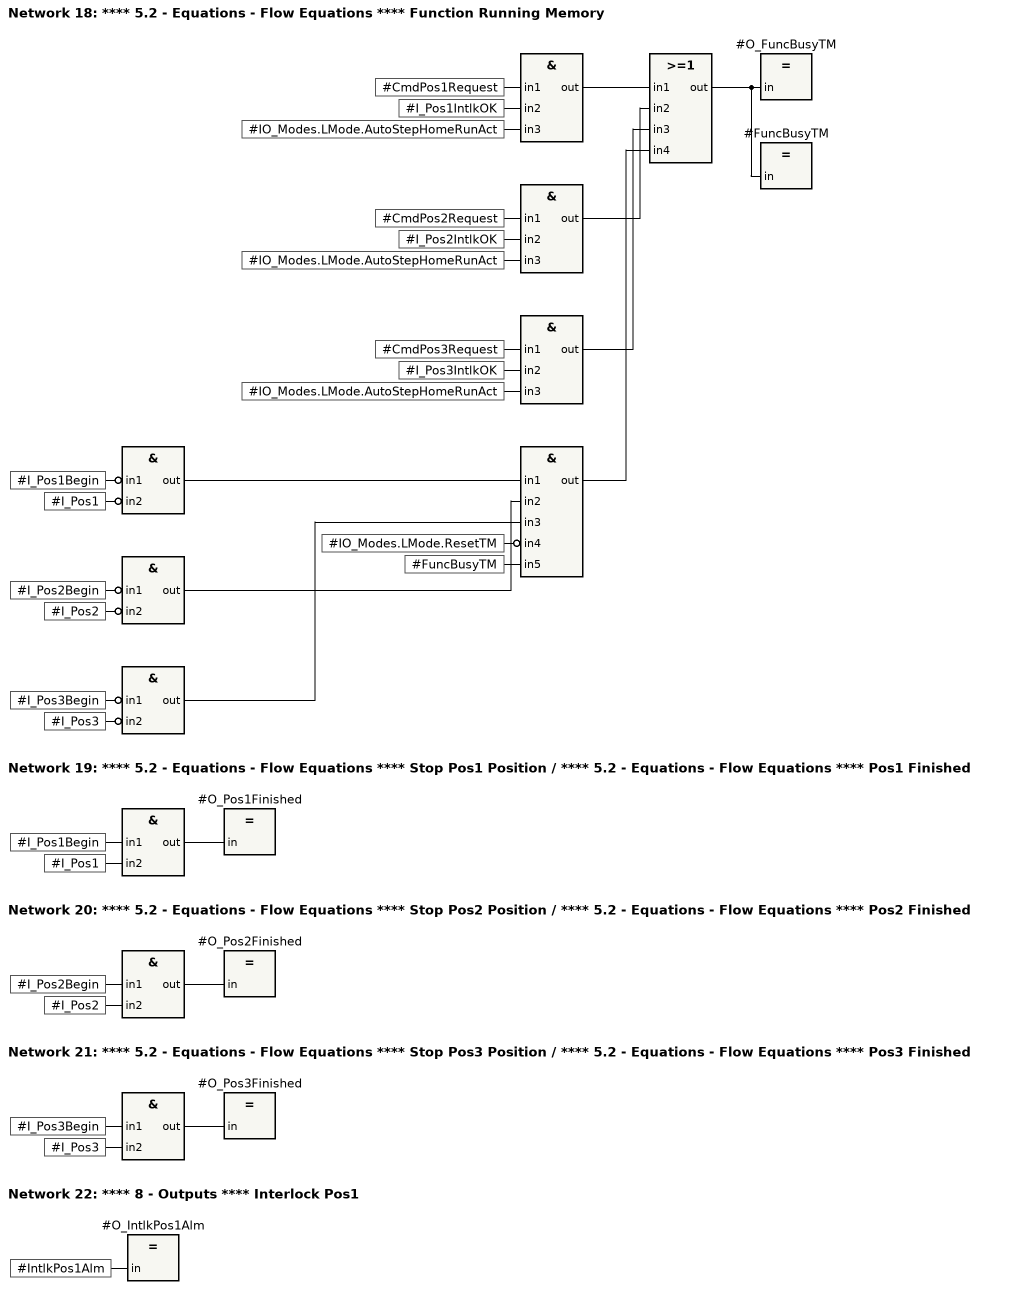
   #O_FuncBusyTM := (#CmdPos1Request AND #I_Pos1IntlkOK AND #IO_Modes.LMode.AutoStepHomeRunAct) OR (#CmdPos2Request AND #I_Pos2IntlkOK AND #IO_Modes.LMode.AutoStepHomeRunAct) OR (#CmdPos3Request AND #I_Pos3IntlkOK AND #IO_Modes.LMode.AutoStepHomeRunAct) OR (NOT #I_Pos1Begin AND NOT #I_Pos1 AND NOT #I_Pos2Begin AND NOT #I_Pos2 AND NOT #I_Pos3Begin AND NOT #I_Pos3 AND NOT #IO_Modes.LMode.ResetTM AND #FuncBusyTM);
   #FuncBusyTM := #O_FuncBusyTM;
END_REGION

REGION Network 19: **** 5.2 - Equations - Flow Equations **** Stop Pos1 Position / **** 5.2 - Equations - Flow Equations **** Pos1 Finished
   // Interlock Pos1
   #O_Pos1Finished := #I_Pos1Begin AND #I_Pos1;
END_REGION

REGION Network 20: **** 5.2 - Equations - Flow Equations **** Stop Pos2 Position / **** 5.2 - Equations - Flow Equations **** Pos2 Finished
   // Interlock Pos2
   #O_Pos2Finished := #I_Pos2Begin AND #I_Pos2;
END_REGION

REGION Network 21: **** 5.2 - Equations - Flow Equations **** Stop Pos3 Position / **** 5.2 - Equations - Flow Equations **** Pos3 Finished
   // Stop Pos3 Position
   #O_Pos3Finished := #I_Pos3Begin AND #I_Pos3;
END_REGION

REGION Network 22: **** 8 - Outputs **** Interlock Pos1
   // Interlock Pos1
   #O_IntlkPos1Alm := #IntlkPos1Alm;
END_REGION

REGION Network 23: **** 8 - Outputs **** Interlock Pos2
   // Interlock Pos2
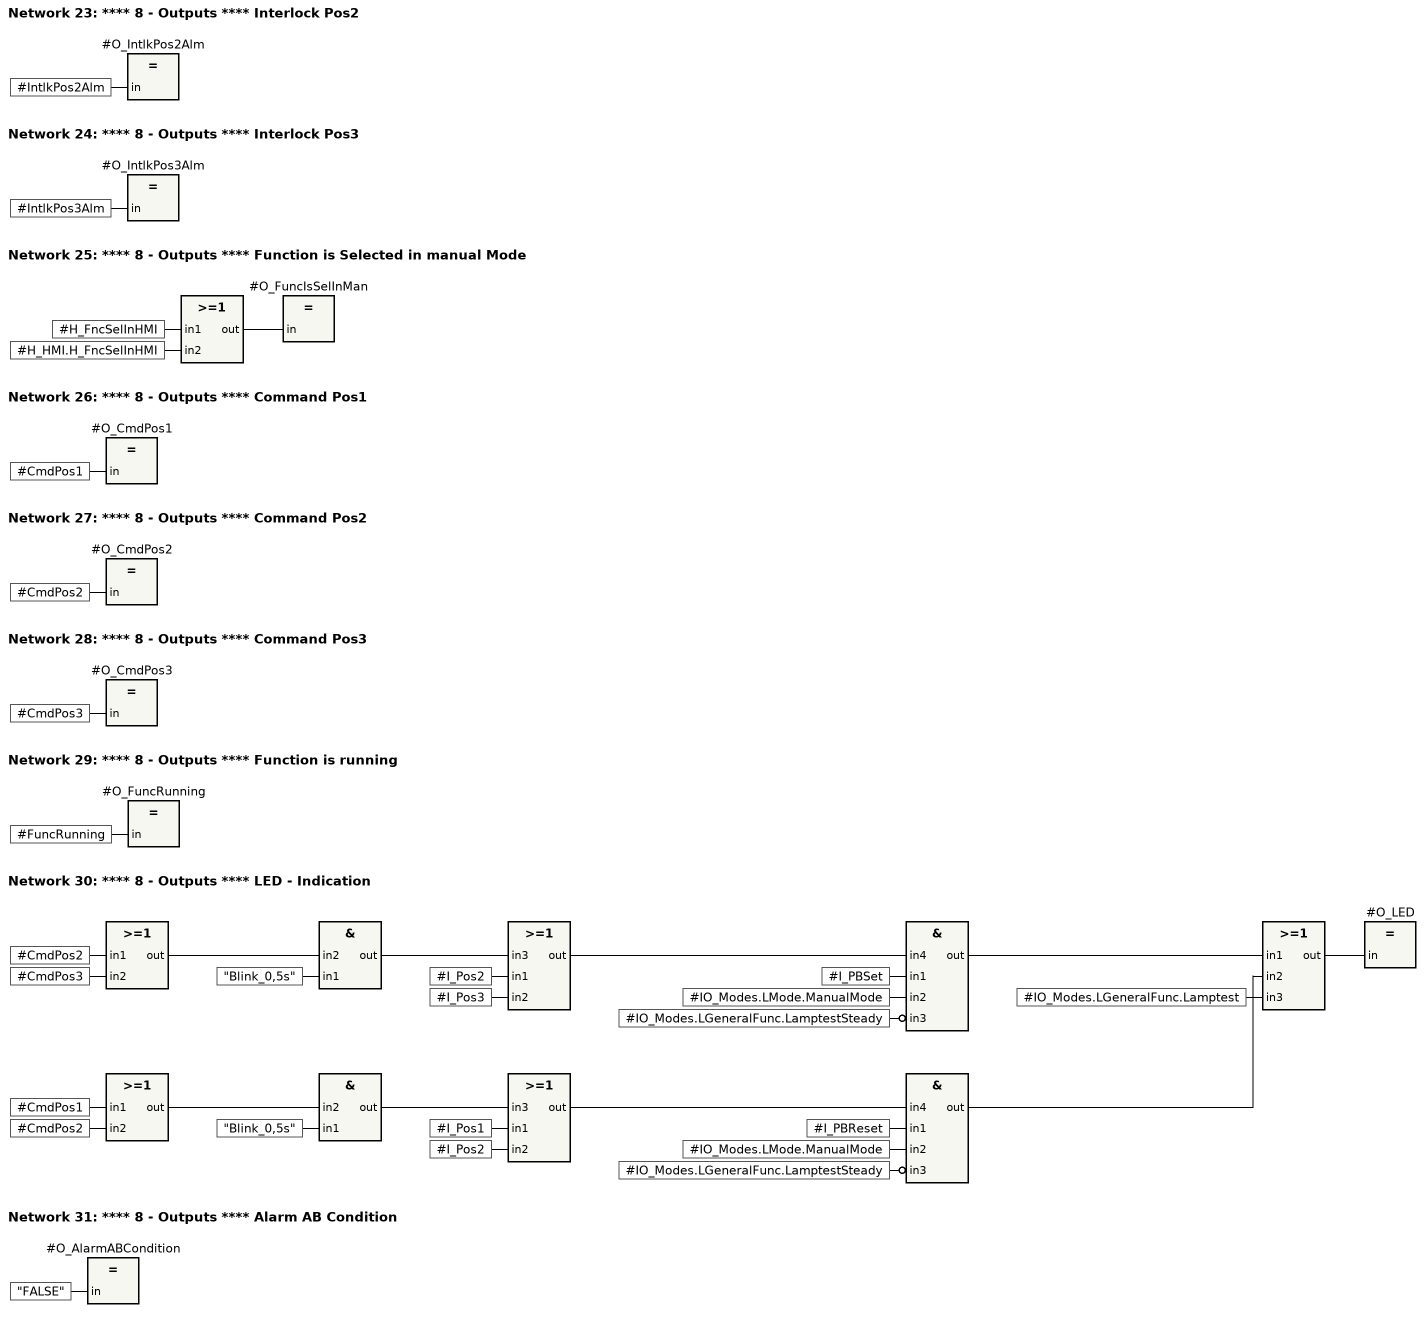
   #O_IntlkPos2Alm := #IntlkPos2Alm;
END_REGION

REGION Network 24: **** 8 - Outputs **** Interlock Pos3
   // Interlock Pos3
   #O_IntlkPos3Alm := #IntlkPos3Alm;
END_REGION

REGION Network 25: **** 8 - Outputs **** Function is Selected in manual Mode
   // Function is Selected in manual Mode
   #O_FuncIsSelInMan := #H_FncSelInHMI OR #H_HMI.H_FncSelInHMI;
END_REGION

REGION Network 26: **** 8 - Outputs **** Command Pos1
   // Command Pos1
   #O_CmdPos1 := #CmdPos1;
END_REGION

REGION Network 27: **** 8 - Outputs **** Command Pos2
   // Command Pos2
   #O_CmdPos2 := #CmdPos2;
END_REGION

REGION Network 28: **** 8 - Outputs **** Command Pos3
   // Command Pos3
   #O_CmdPos3 := #CmdPos3;
END_REGION

REGION Network 29: **** 8 - Outputs **** Function is running
   // Function is running
   #O_FuncRunning := #FuncRunning;
END_REGION

REGION Network 30: **** 8 - Outputs **** LED - Indication
   // LED - Indication
   #O_LED := ((((#CmdPos2 OR #CmdPos3) AND "Blink_0,5s") OR #I_Pos2 OR #I_Pos3) AND #I_PBSet AND #IO_Modes.LMode.ManualMode AND NOT #IO_Modes.LGeneralFunc.LamptestSteady) OR ((((#CmdPos1 OR #CmdPos2) AND "Blink_0,5s") OR #I_Pos1 OR #I_Pos2) AND #I_PBReset AND #IO_Modes.LMode.ManualMode AND NOT #IO_Modes.LGeneralFunc.LamptestSteady) OR #IO_Modes.LGeneralFunc.Lamptest;
END_REGION

REGION Network 31: **** 8 - Outputs **** Alarm AB Condition
   // Alarm AB Condition
   #O_AlarmABCondition := "FALSE";
END_REGION

REGION Network 32: **** 9 - Alarm Summary **** Alarms To Alarm UDT Alarms To Alarm UDT Get Name
   // Alarm / Alarm D
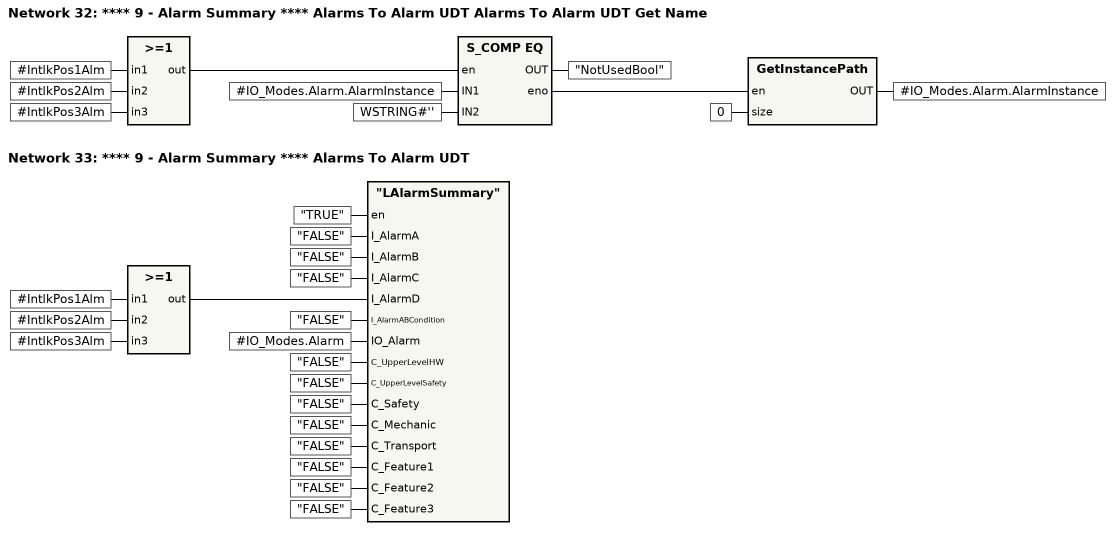
   S_COMP(EN := #IntlkPos1Alm OR #IntlkPos2Alm OR #IntlkPos3Alm,
          IN1 := #IO_Modes.Alarm.AlarmInstance,
          IN2 := WSTRING#'',
          OUT => "NotUsedBool",
          ENO => #_w1);
   IF #_w1 THEN GetInstancePath(size := 0, OUT => #IO_Modes.Alarm.AlarmInstance); END_IF;
END_REGION

REGION Network 33: **** 9 - Alarm Summary **** Alarms To Alarm UDT
   // Alarm / Alarm D
   IF "TRUE" THEN
       "LAlarmSummary"(I_AlarmA := "FALSE",
                       I_AlarmB := "FALSE",
                       I_AlarmC := "FALSE",
                       I_AlarmD := #IntlkPos1Alm OR #IntlkPos2Alm OR #IntlkPos3Alm,
                       I_AlarmABCondition := "FALSE",
                       IO_Alarm := #IO_Modes.Alarm,
                       C_UpperLevelHW := "FALSE",
                       C_UpperLevelSafety := "FALSE",
                       C_Safety := "FALSE",
                       C_Mechanic := "FALSE",
                       C_Transport := "FALSE",
                       C_Feature1 := "FALSE",
                       C_Feature2 := "FALSE",
                       C_Feature3 := "FALSE");
   END_IF;
END_REGION
END_FUNCTION_BLOCK

FUNCTION_BLOCK "L3StopPos"   // FB2188, FBD
TITLE = L3StopPos
{ S7_Optimized_Access := 'TRUE' }
AUTHOR : VCC
FAMILY : Actuator
VERSION : 0.1
// =============================================================================
// This module will be used for a three Position movements.
// It will take care of the Alarms and of the Detections.
// =============================================================================
// stored: AutoNumber false, IsIECCheckEnabled false, IsRetainMemResEnabled false, MemoryReserve 100, SetENOAutomatically False, UDAEnableTagReadback false
   VAR_INPUT
      I_DetPos1 { ExternalAccessible := 'False'; ExternalVisible := 'False'; ExternalWritable := 'False'} : Bool;   // Set detection signal / Pos1 Detection signal
      I_DetPos2 { ExternalAccessible := 'False'; ExternalVisible := 'False'; ExternalWritable := 'False'} : Bool;   // Set detection signal / Pos2 Detection signal
      I_DetPos3 { ExternalAccessible := 'False'; ExternalVisible := 'False'; ExternalWritable := 'False'} : Bool;   // Reset detection signal / Pos3 Detection signal
      I_CmdPos1 { ExternalAccessible := 'False'; ExternalVisible := 'False'; ExternalWritable := 'False'} : Bool;   // function set command / Function Pos1 command
      I_CmdPos2 { ExternalAccessible := 'False'; ExternalVisible := 'False'; ExternalWritable := 'False'} : Bool;   // function set command / Function Pos2 command
      I_CmdPos3 { ExternalAccessible := 'False'; ExternalVisible := 'False'; ExternalWritable := 'False'} : Bool;   // Function reset command / Function Pos3 command
      I_RunPos1 { ExternalAccessible := 'False'; ExternalVisible := 'False'; ExternalWritable := 'False'} : Bool;   // Memory that the Set function is busy / Memory that the Pos1 function is busy
      I_RunPos2 { ExternalAccessible := 'False'; ExternalVisible := 'False'; ExternalWritable := 'False'} : Bool;   // Memory that the Set function is busy / Memory that the Pos2 function is busy
      I_RunPos3 { ExternalAccessible := 'False'; ExternalVisible := 'False'; ExternalWritable := 'False'} : Bool;   // Memory that the Reset function is busy / Memory that the Pos3 function is busy
      I_Pos1IntlkOK { ExternalAccessible := 'False'; ExternalVisible := 'False'; ExternalWritable := 'False'} : Bool;   // Set Interlock / Pos1 Interlock
      I_Pos2IntlkOK { ExternalAccessible := 'False'; ExternalVisible := 'False'; ExternalWritable := 'False'} : Bool;   // Set Interlock / Pos2 Interlock
      I_Pos3IntlkOK { ExternalAccessible := 'False'; ExternalVisible := 'False'; ExternalWritable := 'False'} : Bool;   // Reset Interlock / Pos3 Interlock
      I_SafetyOk { ExternalAccessible := 'False'; ExternalVisible := 'False'; ExternalWritable := 'False'} : Bool;   // Safety Ok
      I_AlarmResetPB { ExternalAccessible := 'False'; ExternalVisible := 'False'; ExternalWritable := 'False'} : Bool := TRUE;   // alarm reset Push Button is activated / Alarm Reset Push Button is Activated
      C_KeepPosition { ExternalAccessible := 'False'; ExternalVisible := 'False'; ExternalWritable := 'False'} : Bool;   // If true, the last position shall be kept ON and checked / If true, the last Position shall be kept ON and checked
      C_EnAlmDet { ExternalAccessible := 'False'; ExternalVisible := 'False'; ExternalWritable := 'False'} : Bool;   // Enable alarm / Enable Alarm
      C_AlarmResetUsed { ExternalAccessible := 'False'; ExternalVisible := 'False'; ExternalWritable := 'False'} : Bool;   // If true, the alarms will be stored untill reseted / If true, the Alarms will be stored untill Reseted
      C_EnAlmOvertime { ExternalAccessible := 'False'; ExternalVisible := 'False'; ExternalWritable := 'False'} : Bool := TRUE;   // Enable Overtime Alarm
      C_RunTimeMaxPos1Warn { ExternalAccessible := 'False'; ExternalVisible := 'False'; ExternalWritable := 'False'} : DInt;   // Maximum Time (ms) that the function may run (create overtime) / Maximum Time (ms) that the function may run (create Overtime)
      C_RunTimeMaxPos1Alm { ExternalAccessible := 'False'; ExternalVisible := 'False'; ExternalWritable := 'False'} : DInt;   // Maximum Time (ms) that the function may run (create overtime) / Maximum Time (ms) that the function may run (create Overtime)
      C_RunTimeMaxPos2Warn { ExternalAccessible := 'False'; ExternalVisible := 'False'; ExternalWritable := 'False'} : DInt;   // Maximum Time (ms) that the function may run (create overtime) / Maximum Time (ms) that the function may run (create Overtime)
      C_RunTimeMaxPos2Alm { ExternalAccessible := 'False'; ExternalVisible := 'False'; ExternalWritable := 'False'} : DInt;   // Maximum Time (ms) that the function may run (create overtime) / Maximum Time (ms) that the function may run (create Overtime)
      C_RunTimeMaxPos3Warn { ExternalAccessible := 'False'; ExternalVisible := 'False'; ExternalWritable := 'False'} : DInt;   // Maximum Time (ms) that the function may run (create overtime) / Maximum Time (ms) that the function may run (create Overtime)
      C_RunTimeMaxPos3Alm { ExternalAccessible := 'False'; ExternalVisible := 'False'; ExternalWritable := 'False'} : DInt;   // Maximum Time (ms) that the function may run (create overtime) / Maximum Time (ms) that the function may run (create Overtime)
      C_TimeAlmFilt { ExternalAccessible := 'False'; ExternalVisible := 'False'; ExternalWritable := 'False'} : DInt := L#2000;   // timer before any actuator alarm will be active (welding..) / timer before any actuator Alarm will be active (welding..)
      C_AlarmSeverityAB { ExternalAccessible := 'False'; ExternalVisible := 'False'; ExternalWritable := 'False'} : Bool;   // Alarm severity
   END_VAR
   VAR_OUTPUT
      O_Pos1 { ExternalAccessible := 'False'; ExternalVisible := 'False'; ExternalWritable := 'False'} : Bool;   // Actuator is in set position / Actuator is in Pos1 Position
      O_Pos2 { ExternalAccessible := 'False'; ExternalVisible := 'False'; ExternalWritable := 'False'} : Bool;   // Actuator is in reset position / Actuator is in Pos2 Position
      O_Pos3 { ExternalAccessible := 'False'; ExternalVisible := 'False'; ExternalWritable := 'False'} : Bool;   // Actuator is in reset position / Actuator is in Pos3 Position
      O_KeepPosPos1Alm { ExternalAccessible := 'False'; ExternalVisible := 'False'; ExternalWritable := 'False'} : Bool;   // Detection Set alarm / Detection Pos1 Alarm
      O_KeepPosPos2Alm { ExternalAccessible := 'False'; ExternalVisible := 'False'; ExternalWritable := 'False'} : Bool;   // Detection Reset alarm / Detection Pos2 Alarm
      O_KeepPosPos3Alm { ExternalAccessible := 'False'; ExternalVisible := 'False'; ExternalWritable := 'False'} : Bool;   // Detection Reset alarm / Detection Pos3 Alarm
      O_MoreThenOneDetAlm { ExternalAccessible := 'False'; ExternalVisible := 'False'; ExternalWritable := 'False'} : Bool;   // Fault condition Both detections ON at the same time / Fault condition More Than One Detections On at the same time
      O_OvtPos1Warn { ExternalAccessible := 'False'; ExternalVisible := 'False'; ExternalWritable := 'False'} : Bool;   // Warning Overtime Set / Warning Overtime Pos1
      O_OvtPos2Warn { ExternalAccessible := 'False'; ExternalVisible := 'False'; ExternalWritable := 'False'} : Bool;   // Warning Overtime Set / Warning Overtime Pos2
      O_OvtPos3Warn { ExternalAccessible := 'False'; ExternalVisible := 'False'; ExternalWritable := 'False'} : Bool;   // Warning Overtime Reset / Warning Overtime Pos3
      O_OvtPos1Alm { ExternalAccessible := 'False'; ExternalVisible := 'False'; ExternalWritable := 'False'} : Bool;   // Alarm Overtime Set / Alarm Overtime Pos1
      O_OvtPos2Alm { ExternalAccessible := 'False'; ExternalVisible := 'False'; ExternalWritable := 'False'} : Bool;   // Alarm Overtime Set / Alarm Overtime Pos2
      O_OvtPos3Alm { ExternalAccessible := 'False'; ExternalVisible := 'False'; ExternalWritable := 'False'} : Bool;   // Alarm Overtime Reset / Alarm Overtime Pos3
      O_ConfigCalibrationAlm { ExternalAccessible := 'False'; ExternalVisible := 'False'; ExternalWritable := 'False'} : Bool;   // Alarm Config/Calibration
      O_CalibrationWarn { ExternalAccessible := 'False'; ExternalVisible := 'False'; ExternalWritable := 'False'} : Bool;   // Warning Calibration
      O_AlarmABCondition { ExternalAccessible := 'False'; ExternalVisible := 'False'; ExternalWritable := 'False'} : Bool;   // Alarm AB condition / Alarm AB Condition
      H_IAnim { ExternalAccessible := 'False'; ExternalVisible := 'False'; ExternalWritable := 'False'} : DWord;   // Icon animation Word / Icon Animation
   END_VAR
   VAR_IN_OUT
      IO_Modes : "Modes";   // Modes
      H_3StopPos : "H_3StopPos";   // Animation
   END_VAR
   VAR
      AlarmReset { ExternalAccessible := 'False'; ExternalVisible := 'False'; ExternalWritable := 'False'} : Bool;   // Alarm Reset Memory
      Pos1PosReq { ExternalAccessible := 'False'; ExternalVisible := 'False'; ExternalWritable := 'False'} : Bool;   // Memorisation of the last set movement / Memorisation of the last Pos1 movement
      Pos2PosReq { ExternalAccessible := 'False'; ExternalVisible := 'False'; ExternalWritable := 'False'} : Bool;   // Memorisation of the last reset movement / Memorisation of the last Pos2 movement
      Pos3PosReq { ExternalAccessible := 'False'; ExternalVisible := 'False'; ExternalWritable := 'False'} : Bool;   // Memorisation of the last reset movement / Memorisation of the last Pos3 movement
      KeepPos1PosOn { ExternalAccessible := 'False'; ExternalVisible := 'False'; ExternalWritable := 'False'} : Bool;   // Check that Set detection is keept on / Check that Pos1 Detection is keept on
      KeepPos2PosOn { ExternalAccessible := 'False'; ExternalVisible := 'False'; ExternalWritable := 'False'} : Bool;   // Check that Set detection is keept on / Check that Pos2 Detection is keept on
      KeepPos3PosOn { ExternalAccessible := 'False'; ExternalVisible := 'False'; ExternalWritable := 'False'} : Bool;   // Check that Set detection is keept on / Check that Pos3 Detection is keept on
      KeepPosPos1StartTimer { ExternalAccessible := 'False'; ExternalVisible := 'False'; ExternalWritable := 'False'} : Bool;   // Detection Set request to start timer / Detection Pos1 Request to start timer
      KeepPosPos2StartTimer { ExternalAccessible := 'False'; ExternalVisible := 'False'; ExternalWritable := 'False'} : Bool;   // Detection Reset request to start timer / Detection Pos2 Request to start timer
      KeepPosPos3StartTimer { ExternalAccessible := 'False'; ExternalVisible := 'False'; ExternalWritable := 'False'} : Bool;   // Detection Reset request to start timer / Detection Pos3 Request to start timer
      MoreThenOneDet { ExternalAccessible := 'False'; ExternalVisible := 'False'; ExternalWritable := 'False'} : Bool;   // Both detections ON at the same time request to start timer / Both Detections ON at the same time Request to start timer
      AlarmFilterStart { ExternalAccessible := 'False'; ExternalVisible := 'False'; ExternalWritable := 'False'} : Bool;   // Alarm filter must be started
      OvtPos1WarnResult { ExternalAccessible := 'False'; ExternalVisible := 'False'; ExternalWritable := 'False'} : Bool;   // Overtime set warning result / Overtime Pos1 warning result
      OvtPos2WarnResult { ExternalAccessible := 'False'; ExternalVisible := 'False'; ExternalWritable := 'False'} : Bool;   // Overtime set warning result / Overtime Pos2 warning result
      OvtPos3WarnResult { ExternalAccessible := 'False'; ExternalVisible := 'False'; ExternalWritable := 'False'} : Bool;   // Overtime reset warning result / Overtime Pos3 warning result
      OvtPos1AlmResult { ExternalAccessible := 'False'; ExternalVisible := 'False'; ExternalWritable := 'False'} : Bool;   // Overtime set alarm result / Overtime Pos1 Alarm result
      OvtPos2AlmResult { ExternalAccessible := 'False'; ExternalVisible := 'False'; ExternalWritable := 'False'} : Bool;   // Overtime reset alarm result / Overtime Pos2 Alarm result
      OvtPos3AlmResult { ExternalAccessible := 'False'; ExternalVisible := 'False'; ExternalWritable := 'False'} : Bool;   // Overtime reset alarm result / Overtime Pos3 Alarm result
      AlmFilterResult { ExternalAccessible := 'False'; ExternalVisible := 'False'; ExternalWritable := 'False'} : Bool;   // Alarm filter result
      MoreThenOneDetAlm { ExternalAccessible := 'False'; ExternalVisible := 'False'; ExternalWritable := 'False'} : Bool;   // Two detection alarm / Pos1 Pos2 Pos3 More Than One Activated
      KeepPos3Alm { ExternalAccessible := 'False'; ExternalVisible := 'False'; ExternalWritable := 'False'} : Bool;   // Keep position Reset alarm / Alarm Keep Position Pos3 Position / Larm Positionsövervakning Pos3 Läge
      KeepPos2Alm { ExternalAccessible := 'False'; ExternalVisible := 'False'; ExternalWritable := 'False'} : Bool;   // Keep position Set alarm / Alarm Keep Position Pos2 Position / Larm Positionsövervakning Pos2 Läge
      KeepPos1Alm { ExternalAccessible := 'False'; ExternalVisible := 'False'; ExternalWritable := 'False'} : Bool;   // Keep position Set alarm / Alarm Keep Position Pos1 Position / Larm Positionsövervakning Pos1 Läge
      OvtPos3Alm { ExternalAccessible := 'False'; ExternalVisible := 'False'; ExternalWritable := 'False'} : Bool;   // Overtime Reset alarm / Overtime Pos3 Alarm
      OvtPos2Alm { ExternalAccessible := 'False'; ExternalVisible := 'False'; ExternalWritable := 'False'} : Bool;   // Overtime Set alarm / Overtime Pos2 Alarm
      OvtPos1Alm { ExternalAccessible := 'False'; ExternalVisible := 'False'; ExternalWritable := 'False'} : Bool;   // Overtime Set alarm / Overtime Pos1 Alarm
      OvtPos3Warn { ExternalAccessible := 'False'; ExternalVisible := 'False'; ExternalWritable := 'False'} : Bool;   // Overtime Reset warning / Overtime Pos3 warning
      OvtPos2Warn { ExternalAccessible := 'False'; ExternalVisible := 'False'; ExternalWritable := 'False'} : Bool;   // Overtime Reset warning / Overtime Pos2 warning
      OvtPos1Warn { ExternalAccessible := 'False'; ExternalVisible := 'False'; ExternalWritable := 'False'} : Bool;   // Overtime Set warning / Overtime Pos1 warning
      ConfigCalibrationAlm { ExternalAccessible := 'False'; ExternalVisible := 'False'; ExternalWritable := 'False'} : Bool;   // Config/Calibration Alarm
      CalibrationWarn { ExternalAccessible := 'False'; ExternalVisible := 'False'; ExternalWritable := 'False'} : Bool;   // Warning Calibration
      Pos1Pos { ExternalAccessible := 'False'; ExternalVisible := 'False'; ExternalWritable := 'False'} : Bool;   // Set position / Pos1 Position
      Pos2Pos { ExternalAccessible := 'False'; ExternalVisible := 'False'; ExternalWritable := 'False'} : Bool;   // Set position / Pos2 Position
      Pos3Pos { ExternalAccessible := 'False'; ExternalVisible := 'False'; ExternalWritable := 'False'} : Bool;   // Reset position / Pos3 Position
      KeepPosPos3AlmCond { ExternalAccessible := 'False'; ExternalVisible := 'False'; ExternalWritable := 'False'} : Bool;   // Keep position reset alarm condition / Keep Position Pos3 Alarm condition
      KeepPosPos2AlmCond { ExternalAccessible := 'False'; ExternalVisible := 'False'; ExternalWritable := 'False'} : Bool;   // Keep position set alarm condition / Keep Position Pos1 Alarm condition
      KeepPosPos1AlmCond { ExternalAccessible := 'False'; ExternalVisible := 'False'; ExternalWritable := 'False'} : Bool;   // Keep position set alarm condition / Keep Position Pos1 Alarm condition
      TwoDetAlmCond { ExternalAccessible := 'False'; ExternalVisible := 'False'; ExternalWritable := 'False'} : Bool;   // Two detector alarm condition / Two or More Detection Alarm condition
      OvtPos3AlmCond { ExternalAccessible := 'False'; ExternalVisible := 'False'; ExternalWritable := 'False'} : Bool;   // Overtime reset alarm condition / Overtime Pos3 Alarm condition
      OvtPos2AlmCond { ExternalAccessible := 'False'; ExternalVisible := 'False'; ExternalWritable := 'False'} : Bool;   // Overtime reset alarm condition / Overtime Pos2 Alarm condition
      OvtPos1AlmCond { ExternalAccessible := 'False'; ExternalVisible := 'False'; ExternalWritable := 'False'} : Bool;   // Overtime set alarm condition / Overtime Pos1 Alarm condition
      Edge { ExternalAccessible := 'False'; ExternalVisible := 'False'; ExternalWritable := 'False'} : Array[1..8] of Bool;   // Edge
      AlarmTimer { ExternalAccessible := 'False'; ExternalVisible := 'False'; ExternalWritable := 'False'} : "LTimer";   // FB
      OvtPos1WarnTimer { ExternalAccessible := 'False'; ExternalVisible := 'False'; ExternalWritable := 'False'} : "LTimer";   // FB
      OvtPos2WarnTimer { ExternalAccessible := 'False'; ExternalVisible := 'False'; ExternalWritable := 'False'} : "LTimer";   // FB
      OvtPos3WarnTimer { ExternalAccessible := 'False'; ExternalVisible := 'False'; ExternalWritable := 'False'} : "LTimer";   // FB
      OvtPos1AlmTimer { ExternalAccessible := 'False'; ExternalVisible := 'False'; ExternalWritable := 'False'} : "LTimer";   // FB
      OvtPos2AlmTimer { ExternalAccessible := 'False'; ExternalVisible := 'False'; ExternalWritable := 'False'} : "LTimer";   // FB
      OvtPos3AlmTimer { ExternalAccessible := 'False'; ExternalVisible := 'False'; ExternalWritable := 'False'} : "LTimer";   // FB
   END_VAR
   VAR RETAIN
      OvtWarnPos1 { ExternalAccessible := 'False'; ExternalVisible := 'False'; ExternalWritable := 'False'} : DInt;   // Alarm Value
      OvtWarnPos2 { ExternalAccessible := 'False'; ExternalVisible := 'False'; ExternalWritable := 'False'} : DInt;   // Alarm Value
      OvtWarnPos3 { ExternalAccessible := 'False'; ExternalVisible := 'False'; ExternalWritable := 'False'} : DInt;   // Alarm Value
      OvtWarnPos1toPos2 { ExternalAccessible := 'False'; ExternalVisible := 'False'; ExternalWritable := 'False'} : DInt;   // Alarm Value
      OvtWarnPos1toPos3 { ExternalAccessible := 'False'; ExternalVisible := 'False'; ExternalWritable := 'False'} : DInt;   // Alarm Value
      OvtWarnPos2toPos3 { ExternalAccessible := 'False'; ExternalVisible := 'False'; ExternalWritable := 'False'} : DInt;   // Alarm Value
      OvtWarnPos2toPos1 { ExternalAccessible := 'False'; ExternalVisible := 'False'; ExternalWritable := 'False'} : DInt;   // Alarm Value
      OvtWarnPos3toPos2 { ExternalAccessible := 'False'; ExternalVisible := 'False'; ExternalWritable := 'False'} : DInt;   // Alarm Value
      OvtWarnPos3toPos1 { ExternalAccessible := 'False'; ExternalVisible := 'False'; ExternalWritable := 'False'} : DInt;   // Alarm Value
      OvtAlarmPos1 { ExternalAccessible := 'False'; ExternalVisible := 'False'; ExternalWritable := 'False'} : DInt;   // Alarm Value
      OvtAlarmPos2 { ExternalAccessible := 'False'; ExternalVisible := 'False'; ExternalWritable := 'False'} : DInt;   // Alarm Value
      OvtAlarmPos3 { ExternalAccessible := 'False'; ExternalVisible := 'False'; ExternalWritable := 'False'} : DInt;   // Alarm Value
      OvtAlarmPos1toPos2 { ExternalAccessible := 'False'; ExternalVisible := 'False'; ExternalWritable := 'False'} : DInt;   // Alarm Value
      OvtAlarmPos1toPos3 { ExternalAccessible := 'False'; ExternalVisible := 'False'; ExternalWritable := 'False'} : DInt;   // Alarm Value
      OvtAlarmPos2toPos3 { ExternalAccessible := 'False'; ExternalVisible := 'False'; ExternalWritable := 'False'} : DInt;   // Alarm Value
      OvtAlarmPos2toPos1 { ExternalAccessible := 'False'; ExternalVisible := 'False'; ExternalWritable := 'False'} : DInt;   // Alarm Value
      OvtAlarmPos3toPos2 { ExternalAccessible := 'False'; ExternalVisible := 'False'; ExternalWritable := 'False'} : DInt;   // Alarm Value
      OvtAlarmPos3toPos1 { ExternalAccessible := 'False'; ExternalVisible := 'False'; ExternalWritable := 'False'} : DInt;   // Alarm Value
      CalibratedPos1toPos2 { ExternalAccessible := 'False'; ExternalVisible := 'False'; ExternalWritable := 'False'} : Bool;   // Calibrated Set
      CalibratedPos1toPos3 { ExternalAccessible := 'False'; ExternalVisible := 'False'; ExternalWritable := 'False'} : Bool;   // Calibrated Reset
      CalibratedPos2toPos3 { ExternalAccessible := 'False'; ExternalVisible := 'False'; ExternalWritable := 'False'} : Bool;   // Calibrated Reset
      CalibratedPos2toPos1 { ExternalAccessible := 'False'; ExternalVisible := 'False'; ExternalWritable := 'False'} : Bool;   // Calibrated Reset
      CalibratedPos3toPos2 { ExternalAccessible := 'False'; ExternalVisible := 'False'; ExternalWritable := 'False'} : Bool;   // Calibrated Reset
      CalibratedPos3toPos1 { ExternalAccessible := 'False'; ExternalVisible := 'False'; ExternalWritable := 'False'} : Bool;   // Calibrated Reset
      MovementPos1toPos3 { ExternalAccessible := 'False'; ExternalVisible := 'False'; ExternalWritable := 'False'} : Bool;   // Calibrated Set
      MovementPos1toPos2 { ExternalAccessible := 'False'; ExternalVisible := 'False'; ExternalWritable := 'False'} : Bool;   // Calibrated Set
      MovementPos3toPos1 { ExternalAccessible := 'False'; ExternalVisible := 'False'; ExternalWritable := 'False'} : Bool;   // Calibrated Set
      MovementPos3toPos2 { ExternalAccessible := 'False'; ExternalVisible := 'False'; ExternalWritable := 'False'} : Bool;   // Calibrated Set
      MovementPos2toPos1 { ExternalAccessible := 'False'; ExternalVisible := 'False'; ExternalWritable := 'False'} : Bool;   // Calibrated Set
      MovementPos2toPos3 { ExternalAccessible := 'False'; ExternalVisible := 'False'; ExternalWritable := 'False'} : Bool;   // Calibrated Set
   END_VAR
   VAR
      AlarmTimeWithConfig { ExternalAccessible := 'False'; ExternalVisible := 'False'; ExternalWritable := 'False'} : Bool;
      AlarmTimeWithCalibration { ExternalAccessible := 'False'; ExternalVisible := 'False'; ExternalWritable := 'False'} : Bool;
      AlmFilterTimerValue { ExternalAccessible := 'False'; ExternalVisible := 'False'; ExternalWritable := 'False'} : DInt;
   END_VAR
   VAR_TEMP
      Cnt : Int;   // Temp
      H_CalibratePos1 : Bool;   // HMI Function
      H_CalibratePos2 : Bool;   // HMI Function
      H_CalibratePos3 : Bool;   // HMI Function
      TempReal : Real;
   END_VAR
   VAR_TEMP   // added for the SCL form of the ladder/FBD networks
      _w1 : Bool;
      _w2 : Bool;
      _w3 : Bool;
      _w4 : Bool;
      _w5 : Bool;
      _w6 : Bool;
      _w7 : Bool;
      _w8 : Bool;
      _w9 : Bool;
      _w10 : Bool;
      _w11 : Bool;
      _w12 : Bool;
      _w13 : Bool;
      _w14 : Bool;
      _w15 : Bool;
   END_VAR
BEGIN

REGION Network 1: **** 1 - Inputs **** HMI Commands
   // Extract the Commands from HMIRobCmd / Extract the Commands from HMI
